KUKA KRL program: EPS_2_25252_SD3A_A_20250910061721.src

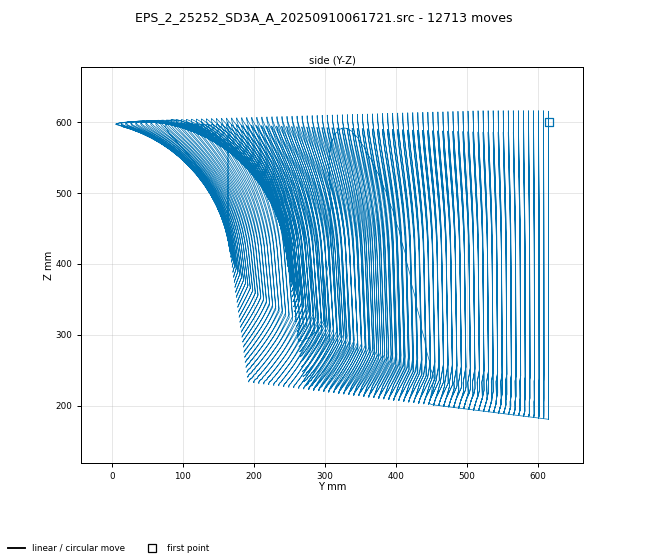
[picture p0: tool path of EPS_2_25252_SD3A_A_20250910061721.src, 12713 of 12715 moves have a stored position in this frame; points joined in program order, loops and branches not executed]
&ACCESS RVP
&REL 4
&COMMENT QRS 19112012
&PARAM EDITMASK = *
DEF PART()
EXT BAS (BAS_COMMAND :IN,REAL :IN )
INT I
BAS (#INITMOV,0 )

;KUKA QRS Post kuka4.cps  Date:22-06-2017 !

File_ID=2824

QRS_PRE_INIT()

;Init var - Until changes are made in qrs_pre_init
Outlet_Square_prg=0
Inlet_1_Square_prg=0
Inlet_2_Square_prg=0
Inlet_3_Square_prg=0
Inlet_4_Square_prg=0
Inlet_5_Square_prg=0

Outlet_1={X 0.000, Y 518.380, Z 433.000, B 0.000, E1 0.000 }
Inlet_1={X 0.000, Y 520.620, Z 403.000, B 0.000, E1 207.000 }
Outlet_1_type=366
Inlet_1_type=366
;QRS#1=Sidecore dimensions
;QRS#2=375-15" PVC SDR 35
;QRS#3=375-15" PVC SDR 35
;QRS#4=
;QRS#5=
;QRS#6=
;QRS#7=
;QRS#8=
;QRS#9=20Y PSX
;QRS#10=20Y PSX
;QRS#11=
;QRS#12=
;QRS#13=
;QRS#14=
;QRS#15=
;QRS#16=1220x127x914 3'
;QRS#17=EPS Height
;QRS#18=616
;QRS#19=*
;QRS#20= UPDATED VERSION 22-06-2017
;QRS#21=*
Outlet_Square=0250
Inlet_1_Square=0250
Inlet_2_Square=0
Inlet_3_Square=0
Inlet_4_Square=0
Inlet_5_Square=0
Mill_Square=1
Outlet_Square_Prg=252
Inlet_1_Square_prg=252

QRS_INIT()

$ADVANCE=5

; T1
PTP {E1 173.576,E2 173.576}
PTP {X 0,Y 615.507,A -85,B 0,C 180,E1 173.576,E2 173.576,E3 0,E4 0,E5 0,E6 0}
QRS_SPEED_INIT()
LIN {X 0,Y 615.507,Z 600,A -85,B 0,C 180,E1 173.576,E2 173.576,E3 0,E4 0,E5 0,E6 0} C_VEL
LIN {X 0,Y 615.507,Z 191.184,A -85,B 0,C 180,E1 173.576,E2 173.576} C_VEL
LIN {X 0,Y 615.507,Z 183.015,A -85,B 0,C 180,E1 173.576,E2 173.576} C_VEL
LIN {X 0,Y 615.486,Z 181.015,A -85,B 0,C 180,E1 173.39,E2 173.39} C_VEL
LIN {X 0,Y 615.462,Z 181.004,A -85,B 0,C 180,E1 170.8,E2 170.8} C_VEL
LIN {X 0,Y 615.46,Z 181.004,A -85,B 0,C 180,E1 168.806,E2 168.806} C_VEL
LIN {X 0,Y 615.457,Z 181.004,A -85,B 0,C 180,E1 166.798,E2 166.798} C_VEL
LIN {X 0,Y 615.453,Z 181.004,A -85,B 0,C 180,E1 164.773,E2 164.773} C_VEL
LIN {X 0,Y 615.448,Z 181.005,A -85,B 0,C 180,E1 162.728,E2 162.728} C_VEL
LIN {X 0,Y 615.442,Z 181.006,A -85,B 0,C 180,E1 160.66,E2 160.66} C_VEL
LIN {X 0,Y 615.437,Z 181.006,A -85,B 0,C 180,E1 158.566,E2 158.566} C_VEL
LIN {X 0,Y 615.45,Z 181.01,A -85,B 0,C 180,E1 155.991,E2 155.991} C_VEL
LIN {X 0,Y 615.495,Z 181.013,A -85,B 0,C 180,E1 153.556,E2 153.556} C_VEL
LIN {X 0,Y 615.489,Z 181.006,A -85,B 0,C 180,E1 151.342,E2 151.342} C_VEL
LIN {X 0,Y 615.45,Z 181.005,A -85,B 0,C 180,E1 148.913,E2 148.913} C_VEL
LIN {X 0,Y 615.432,Z 181.008,A -85,B 0,C 180,E1 146.467,E2 146.467} C_VEL
LIN {X 0,Y 615.445,Z 181.01,A -85,B 0,C 180,E1 144.166,E2 144.166} C_VEL
LIN {X 0,Y 615.47,Z 181.011,A -85,B 0,C 180,E1 141.93,E2 141.93} C_VEL
LIN {X 0,Y 615.488,Z 181.004,A -85,B 0,C 180,E1 139.393,E2 139.393} C_VEL
LIN {X 0,Y 615.434,Z 181.007,A -85,B 0,C 180,E1 136.75,E2 136.75} C_VEL
LIN {X 0,Y 615.467,Z 181.012,A -85,B 0,C 180,E1 133.995,E2 133.995} C_VEL
LIN {X 0,Y 615.448,Z 181.005,A -85,B 0,C 180,E1 131.09,E2 131.09} C_VEL
LIN {X 0,Y 615.433,Z 181.007,A -85,B 0,C 180,E1 128.905,E2 128.905} C_VEL
LIN {X 0,Y 615.44,Z 181.009,A -85,B 0,C 180,E1 126.424,E2 126.424} C_VEL
LIN {X 0,Y 615.477,Z 181.013,A -85,B 0,C 180,E1 124.019,E2 124.019} C_VEL
LIN {X 0,Y 615.439,Z 181.006,A -85,B 0,C 180,E1 121.078,E2 121.078} C_VEL
LIN {X 0,Y 615.434,Z 181.009,A -85,B 0,C 180,E1 118.658,E2 118.658} C_VEL
LIN {X 0,Y 615.499,Z 181.003,A -85,B 0,C 180,E1 115.712,E2 115.712} C_VEL
LIN {X 0,Y 615.474,Z 181.004,A -85,B 0,C 180,E1 113.554,E2 113.554} C_VEL
LIN {X 0,Y 615.456,Z 181.005,A -85,B 0,C 180,E1 111.43,E2 111.43} C_VEL
LIN {X 0,Y 615.447,Z 181.006,A -85,B 0,C 180,E1 109.337,E2 109.337} C_VEL
LIN {X 0,Y 615.441,Z 181.006,A -85,B 0,C 180,E1 107.269,E2 107.269} C_VEL
LIN {X 0,Y 615.437,Z 181.007,A -85,B 0,C 180,E1 105.225,E2 105.225} C_VEL
LIN {X 0,Y 615.435,Z 181.007,A -85,B 0,C 180,E1 103.2,E2 103.2} C_VEL
LIN {X 0,Y 615.432,Z 181.009,A -85,B 0,C 180,E1 100.859,E2 100.859} C_VEL
LIN {X 0,Y 615.452,Z 181.011,A -85,B 0,C 180,E1 98.535,E2 98.535} C_VEL
LIN {X 0,Y 615.493,Z 181.004,A -85,B 0,C 180,E1 95.897,E2 95.897} C_VEL
LIN {X 0,Y 615.433,Z 181.007,A -85,B 0,C 180,E1 93.272,E2 93.272} C_VEL
LIN {X 0,Y 615.433,Z 181.007,A -85,B 0,C 180,E1 91.307,E2 91.307} C_VEL
LIN {X 0,Y 615.434,Z 181.007,A -85,B 0,C 180,E1 89.344,E2 89.344} C_VEL
LIN {X 0,Y 615.429,Z 181.112,A -85,B 0,C 180,E1 87.237,E2 87.237} C_VEL
LIN {X 0,Y 615.455,Z 205.741,A -85,B 0,C 180,E1 84.983,E2 84.983} C_VEL
LIN {X 0,Y 615.489,Z 392.91,A -85,B 0,C 180,E1 82.68,E2 82.68} C_VEL
LIN {X 0,Y 615.492,Z 415.248,A -85,B 0,C 180,E1 82.371,E2 82.371} C_VEL
LIN {X 0,Y 615.494,Z 430.502,A -85,B 0,C 180,E1 82.041,E2 82.041} C_VEL
LIN {X 0,Y 615.492,Z 446.908,A -85,B 0,C 180,E1 81.545,E2 81.545} C_VEL
LIN {X 0,Y 615.491,Z 461.835,A -85,B 0,C 180,E1 80.966,E2 80.966} C_VEL
LIN {X 0,Y 615.492,Z 475.89,A -85,B 0,C 180,E1 80.303,E2 80.303} C_VEL
LIN {X 0,Y 615.498,Z 490.392,A -85,B 0,C 180,E1 79.472,E2 79.472} C_VEL
LIN {X 0,Y 615.497,Z 503.871,A -85,B 0,C 180,E1 78.556,E2 78.556} C_VEL
LIN {X 0,Y 615.495,Z 517.429,A -85,B 0,C 180,E1 77.469,E2 77.469} C_VEL
LIN {X 0,Y 615.496,Z 529.84,A -85,B 0,C 180,E1 76.293,E2 76.293} C_VEL
LIN {X 0,Y 615.489,Z 540.486,A -85,B 0,C 180,E1 75.112,E2 75.112} C_VEL
LIN {X 0,Y 615.495,Z 550.328,A -85,B 0,C 180,E1 73.832,E2 73.832} C_VEL
LIN {X 0,Y 615.493,Z 558.546,A -85,B 0,C 180,E1 72.557,E2 72.557} C_VEL
LIN {X 0,Y 615.489,Z 565.176,A -85,B 0,C 180,E1 71.353,E2 71.353} C_VEL
LIN {X 0,Y 615.496,Z 571.501,A -85,B 0,C 180,E1 69.967,E2 69.967} C_VEL
LIN {X 0,Y 615.484,Z 576.552,A -85,B 0,C 180,E1 68.567,E2 68.567} C_VEL
LIN {X 0,Y 615.484,Z 580.491,A -85,B 0,C 180,E1 67.155,E2 67.155} C_VEL
LIN {X 0,Y 615.487,Z 583.245,A -85,B 0,C 180,E1 65.727,E2 65.727} C_VEL
LIN {X 0,Y 615.5,Z 584.853,A -85,B 0,C 180,E1 64.284,E2 64.284} C_VEL
LIN {X 0,Y 615.493,Z 585.363,A -85,B 0,C 180,E1 62.822,E2 62.822} C_VEL
LIN {X 0,Y 615.486,Z 584.657,A -85,B 0,C 180,E1 61.341,E2 61.341} C_VEL
LIN {X 0,Y 615.494,Z 582.669,A -85,B 0,C 180,E1 59.84,E2 59.84} C_VEL
LIN {X 0,Y 615.491,Z 579.372,A -85,B 0,C 180,E1 58.314,E2 58.314} C_VEL
LIN {X 0,Y 615.487,Z 575.946,A -85,B 0,C 180,E1 57.154,E2 57.154} C_VEL
LIN {X 0,Y 615.489,Z 570.196,A -85,B 0,C 180,E1 55.639,E2 55.639} C_VEL
LIN {X 0,Y 615.495,Z 563.135,A -85,B 0,C 180,E1 54.166,E2 54.166} C_VEL
LIN {X 0,Y 615.491,Z 554.897,A -85,B 0,C 180,E1 52.758,E2 52.758} C_VEL
LIN {X 0,Y 615.495,Z 546.174,A -85,B 0,C 180,E1 51.515,E2 51.515} C_VEL
LIN {X 0,Y 615.494,Z 535.742,A -85,B 0,C 180,E1 50.25,E2 50.25} C_VEL
LIN {X 0,Y 615.492,Z 523.889,A -85,B 0,C 180,E1 49.028,E2 49.028} C_VEL
LIN {X 0,Y 615.493,Z 511.215,A -85,B 0,C 180,E1 47.92,E2 47.92} C_VEL
LIN {X 0,Y 615.494,Z 498.258,A -85,B 0,C 180,E1 46.953,E2 46.953} C_VEL
LIN {X 0,Y 615.496,Z 484.758,A -85,B 0,C 180,E1 46.097,E2 46.097} C_VEL
LIN {X 0,Y 615.491,Z 468.938,A -85,B 0,C 180,E1 45.265,E2 45.265} C_VEL
LIN {X 0,Y 615.495,Z 454.323,A -85,B 0,C 180,E1 44.637,E2 44.637} C_VEL
LIN {X 0,Y 615.491,Z 439.135,A -85,B 0,C 180,E1 44.112,E2 44.112} C_VEL
LIN {X 0,Y 615.496,Z 422.955,A -85,B 0,C 180,E1 43.69,E2 43.69} C_VEL
LIN {X 0,Y 615.491,Z 407.024,A -85,B 0,C 180,E1 43.409,E2 43.409} C_VEL
LIN {X 0,Y 615.482,Z 205.725,A -85,B 0,C 180,E1 40.927,E2 40.927} C_VEL
LIN {X 0,Y 615.492,Z 180.994,A -85,B 0,C 180,E1 38.642,E2 38.642} C_VEL
LIN {X 0,Y 615.493,Z 181.011,A -85,B 0,C 180,E1 35.616,E2 35.616} C_VEL
LIN {X 0,Y 615.472,Z 181.004,A -85,B 0,C 180,E1 33.238,E2 33.238} C_VEL
LIN {X 0,Y 615.48,Z 180.997,A -85,B 0,C 180,E1 30.921,E2 30.921} C_VEL
LIN {X 0,Y 615.486,Z 180.998,A -85,B 0,C 180,E1 28.451,E2 28.451} C_VEL
LIN {X 0,Y 615.477,Z 181.008,A -85,B 0,C 180,E1 25.568,E2 25.568} C_VEL
LIN {X 0,Y 615.49,Z 180.994,A -85,B 0,C 180,E1 22.845,E2 22.845} C_VEL
LIN {X 0,Y 615.486,Z 181.013,A -85,B 0,C 180,E1 20.033,E2 20.033} C_VEL
LIN {X 0,Y 615.469,Z 181.001,A -85,B 0,C 180,E1 17.271,E2 17.271} C_VEL
LIN {X 0,Y 615.487,Z 181,A -85,B 0,C 180,E1 14.549,E2 14.549} C_VEL
LIN {X 0,Y 615.48,Z 181.009,A -85,B 0,C 180,E1 11.861,E2 11.861} C_VEL
LIN {X 0,Y 615.473,Z 180.998,A -85,B 0,C 180,E1 9.199,E2 9.199} C_VEL
LIN {X 0,Y 615.487,Z 181.003,A -85,B 0,C 180,E1 6.557,E2 6.557} C_VEL
LIN {X 0,Y 615.474,Z 181.008,A -85,B 0,C 180,E1 3.929,E2 3.929} C_VEL
LIN {X 0,Y 615.472,Z 180.999,A -85,B 0,C 180,E1 1.309,E2 1.309} C_VEL
LIN {X 0,Y 615.489,Z 181.003,A -85,B 0,C 180,E1 -1.308,E2 -1.308} C_VEL
LIN {X 0,Y 615.473,Z 181.009,A -85,B 0,C 180,E1 -3.928,E2 -3.928} C_VEL
LIN {X 0,Y 615.469,Z 180.999,A -85,B 0,C 180,E1 -6.569,E2 -6.569} C_VEL
LIN {X 0,Y 615.49,Z 181.003,A -85,B 0,C 180,E1 -9.198,E2 -9.198} C_VEL
LIN {X 0,Y 615.469,Z 181.008,A -85,B 0,C 180,E1 -11.861,E2 -11.861} C_VEL
LIN {X 0,Y 615.472,Z 180.999,A -85,B 0,C 180,E1 -14.549,E2 -14.549} C_VEL
LIN {X 0,Y 615.493,Z 181.008,A -85,B 0,C 180,E1 -17.27,E2 -17.27} C_VEL
LIN {X 0,Y 615.454,Z 181.005,A -85,B 0,C 180,E1 -20.034,E2 -20.034} C_VEL
LIN {X 0,Y 615.463,Z 181.001,A -85,B 0,C 180,E1 -22.342,E2 -22.342} C_VEL
LIN {X 0,Y 615.492,Z 181.004,A -85,B 0,C 180,E1 -24.991,E2 -24.991} C_VEL
LIN {X 0,Y 615.453,Z 181.005,A -85,B 0,C 180,E1 -27.916,E2 -27.916} C_VEL
LIN {X 0,Y 615.455,Z 181.002,A -85,B 0,C 180,E1 -30.162,E2 -30.162} C_VEL
LIN {X 0,Y 615.479,Z 180.998,A -85,B 0,C 180,E1 -32.458,E2 -32.458} C_VEL
LIN {X 0,Y 615.492,Z 181.003,A -85,B 0,C 180,E1 -34.814,E2 -34.814} C_VEL
LIN {X 0,Y 615.483,Z 181.011,A -85,B 0,C 180,E1 -37.242,E2 -37.242} C_VEL
LIN {X 0,Y 615.449,Z 181.006,A -85,B 0,C 180,E1 -39.753,E2 -39.753} C_VEL
LIN {X 0,Y 615.478,Z 180.999,A -85,B 0,C 180,E1 -42.353,E2 -42.353} C_VEL
LIN {X 0,Y 615.487,Z 181.012,A -85,B 0,C 180,E1 -45.068,E2 -45.068} C_VEL
LIN {X 0,Y 615.446,Z 181.006,A -85,B 0,C 180,E1 -47.643,E2 -47.643} C_VEL
LIN {X 0,Y 615.476,Z 181,A -85,B 0,C 180,E1 -50.249,E2 -50.249} C_VEL
LIN {X 0,Y 615.472,Z 181.011,A -85,B 0,C 180,E1 -53.065,E2 -53.065} C_VEL
LIN {X 0,Y 615.45,Z 181.008,A -85,B 0,C 180,E1 -55.304,E2 -55.304} C_VEL
LIN {X 0,Y 615.443,Z 181.005,A -85,B 0,C 180,E1 -57.675,E2 -57.675} C_VEL
LIN {X 0,Y 615.482,Z 181.001,A -85,B 0,C 180,E1 -60.206,E2 -60.206} C_VEL
LIN {X 0,Y 615.465,Z 181.01,A -85,B 0,C 180,E1 -62.959,E2 -62.959} C_VEL
LIN {X 0,Y 615.441,Z 181.176,A -85,B 0,C 180,E1 -63.599,E2 -63.599} C_VEL
LIN {X 0,Y 615.497,Z 213.161,A -85,B 0,C 180,E1 -66.217,E2 -66.217} C_VEL
LIN {X 0,Y 615.485,Z 235.002,A -85,B 0,C 180,E1 -67.973,E2 -67.973} C_VEL
LIN {X 0,Y 615.49,Z 442.374,A -85,B 0,C 180,E1 -70.531,E2 -70.531} C_VEL
LIN {X 0,Y 615.493,Z 458.958,A -85,B 0,C 180,E1 -70.878,E2 -70.878} C_VEL
LIN {X 0,Y 615.493,Z 473.906,A -85,B 0,C 180,E1 -71.31,E2 -71.31} C_VEL
LIN {X 0,Y 615.492,Z 489.332,A -85,B 0,C 180,E1 -71.88,E2 -71.88} C_VEL
LIN {X 0,Y 615.493,Z 503.986,A -85,B 0,C 180,E1 -72.557,E2 -72.557} C_VEL
LIN {X 0,Y 615.5,Z 517.82,A -85,B 0,C 180,E1 -73.327,E2 -73.327} C_VEL
LIN {X 0,Y 615.499,Z 532.024,A -85,B 0,C 180,E1 -74.264,E2 -74.264} C_VEL
LIN {X 0,Y 615.495,Z 545.08,A -85,B 0,C 180,E1 -75.281,E2 -75.281} C_VEL
LIN {X 0,Y 615.494,Z 556.202,A -85,B 0,C 180,E1 -76.293,E2 -76.293} C_VEL
LIN {X 0,Y 615.493,Z 567.281,A -85,B 0,C 180,E1 -77.469,E2 -77.469} C_VEL
LIN {X 0,Y 615.495,Z 576.758,A -85,B 0,C 180,E1 -78.639,E2 -78.639} C_VEL
LIN {X 0,Y 615.496,Z 585.957,A -85,B 0,C 180,E1 -79.971,E2 -79.971} C_VEL
LIN {X 0,Y 615.489,Z 594.495,A -85,B 0,C 180,E1 -81.462,E2 -81.462} C_VEL
LIN {X 0,Y 615.491,Z 601.979,A -85,B 0,C 180,E1 -83.101,E2 -83.101} C_VEL
LIN {X 0,Y 615.492,Z 607.737,A -85,B 0,C 180,E1 -84.757,E2 -84.757} C_VEL
LIN {X 0,Y 615.493,Z 611.073,A -85,B 0,C 180,E1 -86.07,E2 -86.07} C_VEL
LIN {X 0,Y 615.485,Z 613.502,A -85,B 0,C 180,E1 -87.381,E2 -87.381} C_VEL
LIN {X 0,Y 615.488,Z 614.869,A -85,B 0,C 180,E1 -88.69,E2 -88.69} C_VEL
LIN {X 0,Y 615.489,Z 615.39,A -85,B 0,C 180,E1 -89.998,E2 -89.998} C_VEL
LIN {X 0,Y 615.488,Z 614.871,A -85,B 0,C 180,E1 -91.307,E2 -91.307} C_VEL
LIN {X 0,Y 615.485,Z 613.507,A -85,B 0,C 180,E1 -92.616,E2 -92.616} C_VEL
LIN {X 0,Y 615.493,Z 611.08,A -85,B 0,C 180,E1 -93.927,E2 -93.927} C_VEL
LIN {X 0,Y 615.492,Z 607.747,A -85,B 0,C 180,E1 -95.239,E2 -95.239} C_VEL
LIN {X 0,Y 615.491,Z 601.986,A -85,B 0,C 180,E1 -96.897,E2 -96.897} C_VEL
LIN {X 0,Y 615.489,Z 594.511,A -85,B 0,C 180,E1 -98.535,E2 -98.535} C_VEL
LIN {X 0,Y 615.496,Z 585.976,A -85,B 0,C 180,E1 -100.026,E2 -100.026} C_VEL
LIN {X 0,Y 615.494,Z 576.781,A -85,B 0,C 180,E1 -101.358,E2 -101.358} C_VEL
LIN {X 0,Y 615.495,Z 567.309,A -85,B 0,C 180,E1 -102.528,E2 -102.528} C_VEL
LIN {X 0,Y 615.496,Z 556.236,A -85,B 0,C 180,E1 -103.703,E2 -103.703} C_VEL
LIN {X 0,Y 615.495,Z 544.141,A -85,B 0,C 180,E1 -104.8,E2 -104.8} C_VEL
LIN {X 0,Y 615.498,Z 530.909,A -85,B 0,C 180,E1 -105.818,E2 -105.818} C_VEL
LIN {X 0,Y 615.5,Z 517.874,A -85,B 0,C 180,E1 -106.669,E2 -106.669} C_VEL
LIN {X 0,Y 615.493,Z 504.053,A -85,B 0,C 180,E1 -107.439,E2 -107.439} C_VEL
LIN {X 0,Y 615.491,Z 489.389,A -85,B 0,C 180,E1 -108.118,E2 -108.118} C_VEL
LIN {X 0,Y 615.493,Z 474.005,A -85,B 0,C 180,E1 -108.687,E2 -108.687} C_VEL
LIN {X 0,Y 615.498,Z 457.273,A -85,B 0,C 180,E1 -109.162,E2 -109.162} C_VEL
LIN {X 0,Y 615.49,Z 441.11,A -85,B 0,C 180,E1 -109.487,E2 -109.487} C_VEL
LIN {X 0,Y 615.485,Z 235.044,A -85,B 0,C 180,E1 -112.024,E2 -112.024} C_VEL
LIN {X 0,Y 615.453,Z 201.645,A -85,B 0,C 180,E1 -114.72,E2 -114.72} C_VEL
LIN {X 0,Y 615.44,Z 181.006,A -85,B 0,C 180,E1 -116.421,E2 -116.421} C_VEL
LIN {X 0,Y 615.441,Z 181.008,A -85,B 0,C 180,E1 -118.657,E2 -118.657} C_VEL
LIN {X 0,Y 615.472,Z 181.011,A -85,B 0,C 180,E1 -121.084,E2 -121.084} C_VEL
LIN {X 0,Y 615.455,Z 181.003,A -85,B 0,C 180,E1 -124.021,E2 -124.021} C_VEL
LIN {X 0,Y 615.438,Z 181.007,A -85,B 0,C 180,E1 -126.425,E2 -126.425} C_VEL
LIN {X 0,Y 615.479,Z 181.011,A -85,B 0,C 180,E1 -129.062,E2 -129.062} C_VEL
LIN {X 0,Y 615.495,Z 181.004,A -85,B 0,C 180,E1 -131.469,E2 -131.469} C_VEL
LIN {X 0,Y 615.441,Z 181.005,A -85,B 0,C 180,E1 -134.149,E2 -134.149} C_VEL
LIN {X 0,Y 615.476,Z 181.011,A -85,B 0,C 180,E1 -136.949,E2 -136.949} C_VEL
LIN {X 0,Y 615.45,Z 181.004,A -85,B 0,C 180,E1 -139.91,E2 -139.91} C_VEL
LIN {X 0,Y 615.444,Z 181.005,A -85,B 0,C 180,E1 -141.988,E2 -141.988} C_VEL
LIN {X 0,Y 615.439,Z 181.008,A -85,B 0,C 180,E1 -144.381,E2 -144.381} C_VEL
LIN {X 0,Y 615.466,Z 181.011,A -85,B 0,C 180,E1 -146.763,E2 -146.763} C_VEL
LIN {X 0,Y 615.491,Z 181.012,A -85,B 0,C 180,E1 -149.081,E2 -149.081} C_VEL
LIN {X 0,Y 615.469,Z 181.003,A -85,B 0,C 180,E1 -151.545,E2 -151.545} C_VEL
LIN {X 0,Y 615.462,Z 181.004,A -85,B 0,C 180,E1 -153.555,E2 -153.555} C_VEL
LIN {X 0,Y 615.437,Z 181.006,A -85,B 0,C 180,E1 -155.993,E2 -155.993} C_VEL
LIN {X 0,Y 615.441,Z 181.005,A -85,B 0,C 180,E1 -157.862,E2 -157.862} C_VEL
LIN {X 0,Y 615.434,Z 181.007,A -85,B 0,C 180,E1 -159.966,E2 -159.966} C_VEL
LIN {X 0,Y 615.478,Z 181.012,A -85,B 0,C 180,E1 -162.73,E2 -162.73} C_VEL
LIN {X 0,Y 615.464,Z 181.003,A -85,B 0,C 180,E1 -165.451,E2 -165.451} C_VEL
LIN {X 0,Y 615.46,Z 181.004,A -85,B 0,C 180,E1 -167.47,E2 -167.47} C_VEL
LIN {X 0,Y 615.457,Z 181.004,A -85,B 0,C 180,E1 -169.473,E2 -169.473} C_VEL
LIN {X 0,Y 615.452,Z 181.005,A -85,B 0,C 180,E1 -171.463,E2 -171.463} C_VEL
LIN {X 0,Y 615.456,Z 181.004,A -85,B 0,C 180,E1 -173.443,E2 -173.443} C_VEL
LIN {X 0,Y 615.456,Z 181.004,A -85,B 0,C 180,E1 -175.416,E2 -175.416} C_VEL
LIN {X 0,Y 615.457,Z 181.004,A -85,B 0,C 180,E1 -177.382,E2 -177.382} C_VEL
LIN {X 0,Y 615.459,Z 181.004,A -85,B 0,C 180,E1 -179.346,E2 -179.346} C_VEL
LIN {X 0,Y 615.46,Z 181.004,A -85,B 0,C 180,E1 -181.309,E2 -181.309} C_VEL
LIN {X 0,Y 615.436,Z 181.008,A -85,B 0,C 180,E1 -183.929,E2 -183.929} C_VEL
LIN {X 0,Y 615.486,Z 181.015,A -85,B 0,C 180,E1 -186.61,E2 -186.61} C_VEL
LIN {X 0,Y 614.795,Z 181.151,A -85,B 0,C 180,E1 -187.156,E2 -187.156} C_VEL
LIN {X 0,Y 611.95,Z 181.566,A -85,B 0,C 180,E1 -188.042,E2 -188.042} C_VEL
LIN {X 0,Y 609.555,Z 181.875,A -85,B 0,C 180,E1 -188.754,E2 -188.754} C_VEL
LIN {X 0,Y 608.517,Z 181.993,A -85,B 0,C 180,E1 -189.304,E2 -189.304} C_VEL
LIN {X 0,Y 608.425,Z 182.003,A -85,B 0,C 180,E1 -189.49,E2 -189.49} C_VEL
LIN {X 0,Y 608.423,Z 182.005,A -85,B 0,C 180,E1 -192.001,E2 -192.001} C_VEL
LIN {X 0,Y 608.465,Z 182.006,A -85,B 0,C 180,E1 -194.721,E2 -194.721} C_VEL
LIN {X 0,Y 608.459,Z 182.005,A -85,B 0,C 180,E1 -196.784,E2 -196.784} C_VEL
LIN {X 0,Y 608.411,Z 182.005,A -85,B 0,C 180,E1 -199.572,E2 -199.572} C_VEL
LIN {X 0,Y 608.429,Z 182.003,A -85,B 0,C 180,E1 -201.693,E2 -201.693} C_VEL
LIN {X 0,Y 608.436,Z 182.01,A -85,B 0,C 180,E1 -204.572,E2 -204.572} C_VEL
LIN {X 0,Y 608.411,Z 182.005,A -85,B 0,C 180,E1 -207.52,E2 -207.52} C_VEL
LIN {X 0,Y 608.431,Z 182.006,A -85,B 0,C 180,E1 -209.973,E2 -209.973} C_VEL
LIN {X 0,Y 608.435,Z 182.004,A -85,B 0,C 180,E1 -212.881,E2 -212.881} C_VEL
LIN {X 0,Y 608.406,Z 182.006,A -85,B 0,C 180,E1 -215.281,E2 -215.281} C_VEL
LIN {X 0,Y 608.439,Z 182.004,A -85,B 0,C 180,E1 -217.749,E2 -217.749} C_VEL
LIN {X 0,Y 608.46,Z 182.009,A -85,B 0,C 180,E1 -220.335,E2 -220.335} C_VEL
LIN {X 0,Y 608.416,Z 182.005,A -85,B 0,C 180,E1 -222.964,E2 -222.964} C_VEL
LIN {X 0,Y 608.411,Z 182.005,A -85,B 0,C 180,E1 -225.204,E2 -225.204} C_VEL
LIN {X 0,Y 608.443,Z 182.007,A -85,B 0,C 180,E1 -227.941,E2 -227.941} C_VEL
LIN {X 0,Y 608.42,Z 182.006,A -85,B 0,C 180,E1 -230.709,E2 -230.709} C_VEL
LIN {X 0,Y 608.407,Z 182.005,A -85,B 0,C 180,E1 -233.085,E2 -233.085} C_VEL
LIN {X 0,Y 608.432,Z 182.004,A -85,B 0,C 180,E1 -235.532,E2 -235.532} C_VEL
LIN {X 0,Y 608.445,Z 182.008,A -85,B 0,C 180,E1 -237.908,E2 -237.908} C_VEL
LIN {X 0,Y 608.48,Z 182.004,A -85,B 0,C 180,E1 -240.224,E2 -240.224} C_VEL
LIN {X 0,Y 608.403,Z 182.006,A -85,B 0,C 180,E1 -243.226,E2 -243.226} C_VEL
LIN {X 0,Y 608.422,Z 182.006,A -85,B 0,C 180,E1 -245.43,E2 -245.43} C_VEL
LIN {X 0,Y 608.45,Z 182.005,A -85,B 0,C 180,E1 -248.31,E2 -248.31} C_VEL
LIN {X 0,Y 608.427,Z 182.003,A -85,B 0,C 180,E1 -251.132,E2 -251.132} C_VEL
LIN {X 0,Y 608.453,Z 182.011,A -85,B 0,C 180,E1 -253.908,E2 -253.908} C_VEL
LIN {X 0,Y 608.43,Z 182.003,A -85,B 0,C 180,E1 -256.645,E2 -256.645} C_VEL
LIN {X 0,Y 608.425,Z 182.006,A -85,B 0,C 180,E1 -259.352,E2 -259.352} C_VEL
LIN {X 0,Y 608.473,Z 182.005,A -85,B 0,C 180,E1 -262.035,E2 -262.035} C_VEL
LIN {X 0,Y 608.421,Z 182.004,A -85,B 0,C 180,E1 -264.7,E2 -264.7} C_VEL
LIN {X 0,Y 608.444,Z 182.005,A -85,B 0,C 180,E1 -267.354,E2 -267.354} C_VEL
LIN {X 0,Y 608.477,Z 182.004,A -85,B 0,C 180,E1 -270.002,E2 -270.002} C_VEL
LIN {X 0,Y 608.436,Z 182.197,A -85,B 0,C 180,E1 -272.567,E2 -272.567} C_VEL
LIN {X 0,Y 608.717,Z 193.625,A -85,B 0,C 180,E1 -273.642,E2 -273.642} C_VEL
LIN {X 0,Y 608.636,Z 205.796,A -85,B 0,C 180,E1 -274.762,E2 -274.762} C_VEL
LIN {X 0,Y 608.876,Z 210.931,A -85,B 0,C 180,E1 -274.843,E2 -274.843} C_VEL
LIN {X 0,Y 608.815,Z 411.348,A -85,B 0,C 180,E1 -277.338,E2 -277.338} C_VEL
LIN {X 0,Y 608.775,Z 427.683,A -85,B 0,C 180,E1 -277.672,E2 -277.672} C_VEL
LIN {X 0,Y 608.754,Z 443.666,A -85,B 0,C 180,E1 -278.132,E2 -278.132} C_VEL
LIN {X 0,Y 608.703,Z 459.382,A -85,B 0,C 180,E1 -278.717,E2 -278.717} C_VEL
LIN {X 0,Y 608.66,Z 475.413,A -85,B 0,C 180,E1 -279.472,E2 -279.472} C_VEL
LIN {X 0,Y 608.629,Z 490.001,A -85,B 0,C 180,E1 -280.312,E2 -280.312} C_VEL
LIN {X 0,Y 608.585,Z 503.661,A -85,B 0,C 180,E1 -281.246,E2 -281.246} C_VEL
LIN {X 0,Y 608.544,Z 517.201,A -85,B 0,C 180,E1 -282.338,E2 -282.338} C_VEL
LIN {X 0,Y 608.497,Z 529.711,A -85,B 0,C 180,E1 -283.527,E2 -283.527} C_VEL
LIN {X 0,Y 608.486,Z 540.445,A -85,B 0,C 180,E1 -284.721,E2 -284.721} C_VEL
LIN {X 0,Y 608.458,Z 550.929,A -85,B 0,C 180,E1 -286.095,E2 -286.095} C_VEL
LIN {X 0,Y 608.469,Z 559.727,A -85,B 0,C 180,E1 -287.477,E2 -287.477} C_VEL
LIN {X 0,Y 608.443,Z 567.104,A -85,B 0,C 180,E1 -288.871,E2 -288.871} C_VEL
LIN {X 0,Y 608.438,Z 573.211,A -85,B 0,C 180,E1 -290.276,E2 -290.276} C_VEL
LIN {X 0,Y 608.426,Z 578.09,A -85,B 0,C 180,E1 -291.694,E2 -291.694} C_VEL
LIN {X 0,Y 608.427,Z 581.751,A -85,B 0,C 180,E1 -293.126,E2 -293.126} C_VEL
LIN {X 0,Y 608.406,Z 584.315,A -85,B 0,C 180,E1 -294.574,E2 -294.574} C_VEL
LIN {X 0,Y 608.42,Z 585.7,A -85,B 0,C 180,E1 -296.037,E2 -296.037} C_VEL
LIN {X 0,Y 608.425,Z 585.894,A -85,B 0,C 180,E1 -297.52,E2 -297.52} C_VEL
LIN {X 0,Y 608.407,Z 584.897,A -85,B 0,C 180,E1 -299.024,E2 -299.024} C_VEL
LIN {X 0,Y 608.43,Z 582.651,A -85,B 0,C 180,E1 -300.548,E2 -300.548} C_VEL
LIN {X 0,Y 608.417,Z 578.946,A -85,B 0,C 180,E1 -302.098,E2 -302.098} C_VEL
LIN {X 0,Y 608.425,Z 573.535,A -85,B 0,C 180,E1 -303.727,E2 -303.727} C_VEL
LIN {X 0,Y 608.43,Z 566.815,A -85,B 0,C 180,E1 -305.279,E2 -305.279} C_VEL
LIN {X 0,Y 608.471,Z 559.156,A -85,B 0,C 180,E1 -306.708,E2 -306.708} C_VEL
LIN {X 0,Y 608.48,Z 550.942,A -85,B 0,C 180,E1 -307.993,E2 -307.993} C_VEL
LIN {X 0,Y 608.483,Z 541.012,A -85,B 0,C 180,E1 -309.298,E2 -309.298} C_VEL
LIN {X 0,Y 608.508,Z 530.16,A -85,B 0,C 180,E1 -310.516,E2 -310.516} C_VEL
LIN {X 0,Y 608.547,Z 518.193,A -85,B 0,C 180,E1 -311.665,E2 -311.665} C_VEL
LIN {X 0,Y 608.573,Z 505.702,A -85,B 0,C 180,E1 -312.693,E2 -312.693} C_VEL
LIN {X 0,Y 608.611,Z 492.473,A -85,B 0,C 180,E1 -313.624,E2 -313.624} C_VEL
LIN {X 0,Y 608.643,Z 478.411,A -85,B 0,C 180,E1 -314.455,E2 -314.455} C_VEL
LIN {X 0,Y 608.689,Z 462.722,A -85,B 0,C 180,E1 -315.225,E2 -315.225} C_VEL
LIN {X 0,Y 608.73,Z 446.825,A -85,B 0,C 180,E1 -315.852,E2 -315.852} C_VEL
LIN {X 0,Y 608.768,Z 430.544,A -85,B 0,C 180,E1 -316.349,E2 -316.349} C_VEL
LIN {X 0,Y 608.801,Z 413.508,A -85,B 0,C 180,E1 -316.717,E2 -316.717} C_VEL
LIN {X 0,Y 608.821,Z 376.219,A -85,B 0,C 180,E1 -317.2,E2 -317.2} C_VEL
LIN {X 0,Y 608.878,Z 206.999,A -85,B 0,C 180,E1 -319.296,E2 -319.296} C_VEL
LIN {X 0,Y 608.692,Z 205.634,A -85,B 0,C 180,E1 -319.341,E2 -319.341} C_VEL
LIN {X 0,Y 608.709,Z 183.074,A -85,B 0,C 180,E1 -321.429,E2 -321.429} C_VEL
LIN {X 0,Y 608.463,Z 182.001,A -85,B 0,C 180,E1 -321.552,E2 -321.552} C_VEL
LIN {X 0,Y 608.462,Z 182.004,A -85,B 0,C 180,E1 -323.952,E2 -323.952} C_VEL
LIN {X 0,Y 608.45,Z 182.01,A -85,B 0,C 180,E1 -326.328,E2 -326.328} C_VEL
LIN {X 0,Y 608.444,Z 182.004,A -85,B 0,C 180,E1 -328.732,E2 -328.732} C_VEL
LIN {X 0,Y 608.474,Z 181.998,A -85,B 0,C 180,E1 -331.379,E2 -331.379} C_VEL
LIN {X 0,Y 608.469,Z 182.006,A -85,B 0,C 180,E1 -334.279,E2 -334.279} C_VEL
LIN {X 0,Y 608.449,Z 182.001,A -85,B 0,C 180,E1 -336.876,E2 -336.876} C_VEL
LIN {X 0,Y 608.462,Z 182.004,A -85,B 0,C 180,E1 -339.725,E2 -339.725} C_VEL
LIN {X 0,Y 608.444,Z 182.003,A -85,B 0,C 180,E1 -342.523,E2 -342.523} C_VEL
LIN {X 0,Y 608.471,Z 181.999,A -85,B 0,C 180,E1 -345.279,E2 -345.279} C_VEL
LIN {X 0,Y 608.457,Z 182.009,A -85,B 0,C 180,E1 -348,E2 -348} C_VEL
LIN {X 0,Y 608.458,Z 182,A -85,B 0,C 180,E1 -350.694,E2 -350.694} C_VEL
LIN {X 0,Y 608.474,Z 182.001,A -85,B 0,C 180,E1 -353.367,E2 -353.367} C_VEL
LIN {X 0,Y 608.444,Z 182.007,A -85,B 0,C 180,E1 -356.026,E2 -356.026} C_VEL
LIN {X 0,Y 608.456,Z 181.999,A -85,B 0,C 180,E1 -358.676,E2 -358.676} C_VEL
LIN {X 0,Y 608.471,Z 182.002,A -85,B 0,C 180,E1 -361.323,E2 -361.323} C_VEL
LIN {X 0,Y 608.441,Z 182.006,A -85,B 0,C 180,E1 -363.974,E2 -363.974} C_VEL
LIN {X 0,Y 608.454,Z 182,A -85,B 0,C 180,E1 -366.632,E2 -366.632} C_VEL
LIN {X 0,Y 608.47,Z 182.004,A -85,B 0,C 180,E1 -369.305,E2 -369.305} C_VEL
LIN {X 0,Y 608.446,Z 182.004,A -85,B 0,C 180,E1 -372,E2 -372} C_VEL
LIN {X 0,Y 608.466,Z 181.999,A -85,B 0,C 180,E1 -374.72,E2 -374.72} C_VEL
LIN {X 0,Y 608.449,Z 182.01,A -85,B 0,C 180,E1 -377.476,E2 -377.476} C_VEL
LIN {X 0,Y 608.44,Z 182.001,A -85,B 0,C 180,E1 -380.275,E2 -380.275} C_VEL
LIN {X 0,Y 608.454,Z 182,A -85,B 0,C 180,E1 -382.476,E2 -382.476} C_VEL
LIN {X 0,Y 608.445,Z 182.012,A -85,B 0,C 180,E1 -385.301,E2 -385.301} C_VEL
LIN {X 0,Y 608.437,Z 182.008,A -85,B 0,C 180,E1 -387.518,E2 -387.518} C_VEL
LIN {X 0,Y 608.438,Z 182.002,A -85,B 0,C 180,E1 -389.967,E2 -389.967} C_VEL
LIN {X 0,Y 608.455,Z 182.001,A -85,B 0,C 180,E1 -392.522,E2 -392.522} C_VEL
LIN {X 0,Y 608.428,Z 182.011,A -85,B 0,C 180,E1 -395.278,E2 -395.278} C_VEL
LIN {X 0,Y 608.448,Z 182.002,A -85,B 0,C 180,E1 -397.747,E2 -397.747} C_VEL
LIN {X 0,Y 608.439,Z 182.002,A -85,B 0,C 180,E1 -400.328,E2 -400.328} C_VEL
LIN {X 0,Y 608.46,Z 182.004,A -85,B 0,C 180,E1 -403.308,E2 -403.308} C_VEL
LIN {X 0,Y 608.447,Z 182.001,A -85,B 0,C 180,E1 -406.128,E2 -406.128} C_VEL
LIN {X 0,Y 608.457,Z 182.009,A -85,B 0,C 180,E1 -408.823,E2 -408.823} C_VEL
LIN {X 0,Y 608.421,Z 182.006,A -85,B 0,C 180,E1 -411.408,E2 -411.408} C_VEL
LIN {X 0,Y 608.438,Z 182.002,A -85,B 0,C 180,E1 -413.955,E2 -413.955} C_VEL
LIN {X 0,Y 608.467,Z 182.002,A -85,B 0,C 180,E1 -416.329,E2 -416.329} C_VEL
LIN {X 0,Y 608.445,Z 182.012,A -85,B 0,C 180,E1 -418.732,E2 -418.732} C_VEL
LIN {X 0,Y 608.436,Z 182.004,A -85,B 0,C 180,E1 -421.386,E2 -421.386} C_VEL
LIN {X 0,Y 608.458,Z 182.142,A -85,B 0,C 180,E1 -423.353,E2 -423.353} C_VEL
LIN {X 0,Y 608.799,Z 186.144,A -85,B 0,C 180,E1 -423.704,E2 -423.704} C_VEL
LIN {X 0,Y 608.749,Z 219.268,A -85,B 0,C 180,E1 -426.437,E2 -426.437} C_VEL
LIN {X 0,Y 608.705,Z 235.002,A -85,B 0,C 180,E1 -427.715,E2 -427.715} C_VEL
LIN {X 0,Y 608.907,Z 243.7,A -85,B 0,C 180,E1 -427.834,E2 -427.834} C_VEL
LIN {X 0,Y 608.804,Z 442.373,A -85,B 0,C 180,E1 -430.309,E2 -430.309} C_VEL
LIN {X 0,Y 608.795,Z 458.96,A -85,B 0,C 180,E1 -430.659,E2 -430.659} C_VEL
LIN {X 0,Y 608.744,Z 475.202,A -85,B 0,C 180,E1 -431.139,E2 -431.139} C_VEL
LIN {X 0,Y 608.688,Z 491.193,A -85,B 0,C 180,E1 -431.752,E2 -431.752} C_VEL
LIN {X 0,Y 608.681,Z 505.712,A -85,B 0,C 180,E1 -432.443,E2 -432.443} C_VEL
LIN {X 0,Y 608.633,Z 520.92,A -85,B 0,C 180,E1 -433.323,E2 -433.323} C_VEL
LIN {X 0,Y 608.574,Z 534.354,A -85,B 0,C 180,E1 -434.252,E2 -434.252} C_VEL
LIN {X 0,Y 608.548,Z 547.055,A -85,B 0,C 180,E1 -435.28,E2 -435.28} C_VEL
LIN {X 0,Y 608.496,Z 559.624,A -85,B 0,C 180,E1 -436.473,E2 -436.473} C_VEL
LIN {X 0,Y 608.47,Z 570.321,A -85,B 0,C 180,E1 -437.661,E2 -437.661} C_VEL
LIN {X 0,Y 608.474,Z 580.866,A -85,B 0,C 180,E1 -439.041,E2 -439.041} C_VEL
LIN {X 0,Y 608.466,Z 589.276,A -85,B 0,C 180,E1 -440.357,E2 -440.357} C_VEL
LIN {X 0,Y 608.452,Z 596.479,A -85,B 0,C 180,E1 -441.697,E2 -441.697} C_VEL
LIN {X 0,Y 608.438,Z 602.463,A -85,B 0,C 180,E1 -443.032,E2 -443.032} C_VEL
LIN {X 0,Y 608.435,Z 608.241,A -85,B 0,C 180,E1 -444.696,E2 -444.696} C_VEL
LIN {X 0,Y 608.43,Z 611.629,A -85,B 0,C 180,E1 -446.024,E2 -446.024} C_VEL
LIN {X 0,Y 608.412,Z 614.083,A -85,B 0,C 180,E1 -447.35,E2 -447.35} C_VEL
LIN {X 0,Y 608.441,Z 615.476,A -85,B 0,C 180,E1 -448.675,E2 -448.675} C_VEL
LIN {X 0,Y 608.429,Z 616,A -85,B 0,C 180,E1 -449.998,E2 -449.998} C_VEL
LIN {X 0,Y 608.44,Z 615.478,A -85,B 0,C 180,E1 -451.322,E2 -451.322} C_VEL
LIN {X 0,Y 608.412,Z 614.088,A -85,B 0,C 180,E1 -452.647,E2 -452.647} C_VEL
LIN {X 0,Y 608.43,Z 611.636,A -85,B 0,C 180,E1 -453.972,E2 -453.972} C_VEL
LIN {X 0,Y 608.435,Z 608.251,A -85,B 0,C 180,E1 -455.3,E2 -455.3} C_VEL
LIN {X 0,Y 608.436,Z 602.476,A -85,B 0,C 180,E1 -456.964,E2 -456.964} C_VEL
LIN {X 0,Y 608.443,Z 594.867,A -85,B 0,C 180,E1 -458.634,E2 -458.634} C_VEL
LIN {X 0,Y 608.461,Z 586.257,A -85,B 0,C 180,E1 -460.143,E2 -460.143} C_VEL
LIN {X 0,Y 608.466,Z 576.983,A -85,B 0,C 180,E1 -461.491,E2 -461.491} C_VEL
LIN {X 0,Y 608.49,Z 567.44,A -85,B 0,C 180,E1 -462.674,E2 -462.674} C_VEL
LIN {X 0,Y 608.524,Z 555.952,A -85,B 0,C 180,E1 -463.897,E2 -463.897} C_VEL
LIN {X 0,Y 608.552,Z 544.169,A -85,B 0,C 180,E1 -464.973,E2 -464.973} C_VEL
LIN {X 0,Y 608.597,Z 530.916,A -85,B 0,C 180,E1 -466.002,E2 -466.002} C_VEL
LIN {X 0,Y 608.616,Z 517.877,A -85,B 0,C 180,E1 -466.863,E2 -466.863} C_VEL
LIN {X 0,Y 608.677,Z 502.309,A -85,B 0,C 180,E1 -467.728,E2 -467.728} C_VEL
LIN {X 0,Y 608.711,Z 487.407,A -85,B 0,C 180,E1 -468.409,E2 -468.409} C_VEL
LIN {X 0,Y 608.736,Z 471.42,A -85,B 0,C 180,E1 -468.989,E2 -468.989} C_VEL
LIN {X 0,Y 608.792,Z 455.45,A -85,B 0,C 180,E1 -469.425,E2 -469.425} C_VEL
LIN {X 0,Y 608.807,Z 439.604,A -85,B 0,C 180,E1 -469.732,E2 -469.732} C_VEL
LIN {X 0,Y 608.91,Z 236.821,A -85,B 0,C 180,E1 -472.252,E2 -472.252} C_VEL
LIN {X 0,Y 608.719,Z 234.768,A -85,B 0,C 180,E1 -472.304,E2 -472.304} C_VEL
LIN {X 0,Y 608.772,Z 201.645,A -85,B 0,C 180,E1 -475.01,E2 -475.01} C_VEL
LIN {X 0,Y 608.807,Z 183.979,A -85,B 0,C 180,E1 -476.477,E2 -476.477} C_VEL
LIN {X 0,Y 608.415,Z 182.009,A -85,B 0,C 180,E1 -476.68,E2 -476.68} C_VEL
LIN {X 0,Y 608.465,Z 182.002,A -85,B 0,C 180,E1 -479.777,E2 -479.777} C_VEL
LIN {X 0,Y 608.419,Z 182.004,A -85,B 0,C 180,E1 -482.517,E2 -482.517} C_VEL
LIN {X 0,Y 608.448,Z 182.005,A -85,B 0,C 180,E1 -484.906,E2 -484.906} C_VEL
LIN {X 0,Y 608.448,Z 182.003,A -85,B 0,C 180,E1 -487.744,E2 -487.744} C_VEL
LIN {X 0,Y 608.41,Z 182.005,A -85,B 0,C 180,E1 -490.325,E2 -490.325} C_VEL
LIN {X 0,Y 608.437,Z 182.009,A -85,B 0,C 180,E1 -492.957,E2 -492.957} C_VEL
LIN {X 0,Y 608.43,Z 182.004,A -85,B 0,C 180,E1 -495.734,E2 -495.734} C_VEL
LIN {X 0,Y 608.431,Z 182.003,A -85,B 0,C 180,E1 -497.936,E2 -497.936} C_VEL
LIN {X 0,Y 608.453,Z 182.004,A -85,B 0,C 180,E1 -500.699,E2 -500.699} C_VEL
LIN {X 0,Y 608.455,Z 182.01,A -85,B 0,C 180,E1 -503.085,E2 -503.085} C_VEL
LIN {X 0,Y 608.461,Z 182.002,A -85,B 0,C 180,E1 -505.531,E2 -505.531} C_VEL
LIN {X 0,Y 608.435,Z 182.002,A -85,B 0,C 180,E1 -507.904,E2 -507.904} C_VEL
LIN {X 0,Y 608.42,Z 182.004,A -85,B 0,C 180,E1 -510.218,E2 -510.218} C_VEL
LIN {X 0,Y 608.47,Z 182.005,A -85,B 0,C 180,E1 -512.787,E2 -512.787} C_VEL
LIN {X 0,Y 608.436,Z 182.002,A -85,B 0,C 180,E1 -515.848,E2 -515.848} C_VEL
LIN {X 0,Y 608.434,Z 182.004,A -85,B 0,C 180,E1 -518.307,E2 -518.307} C_VEL
LIN {X 0,Y 608.45,Z 182.004,A -85,B 0,C 180,E1 -521.278,E2 -521.278} C_VEL
LIN {X 0,Y 608.419,Z 182.004,A -85,B 0,C 180,E1 -523.905,E2 -523.905} C_VEL
LIN {X 0,Y 608.455,Z 182.007,A -85,B 0,C 180,E1 -526.644,E2 -526.644} C_VEL
LIN {X 0,Y 608.445,Z 182.003,A -85,B 0,C 180,E1 -529.35,E2 -529.35} C_VEL
LIN {X 0,Y 608.432,Z 182.003,A -85,B 0,C 180,E1 -532.033,E2 -532.033} C_VEL
LIN {X 0,Y 608.467,Z 182.008,A -85,B 0,C 180,E1 -534.698,E2 -534.698} C_VEL
LIN {X 0,Y 608.449,Z 182.001,A -85,B 0,C 180,E1 -537.352,E2 -537.352} C_VEL
LIN {X 0,Y 608.429,Z 182.004,A -85,B 0,C 180,E1 -540,E2 -540} C_VEL
LIN {X 0,Y 608.473,Z 182.008,A -85,B 0,C 180,E1 -542.648,E2 -542.648} C_VEL
LIN {X 0,Y 608.438,Z 182.003,A -85,B 0,C 180,E1 -545.302,E2 -545.302} C_VEL
LIN {X 0,Y 608.452,Z 182.001,A -85,B 0,C 180,E1 -547.3,E2 -547.3} C_VEL
LIN {X 0,Y 608.425,Z 182.003,A -85,B 0,C 180,E1 -549.49,E2 -549.49} C_VEL
LIN {X 0,Y 607.739,Z 182.092,A -85,B 0,C 180,E1 -550.043,E2 -550.043} C_VEL
LIN {X 0,Y 604.879,Z 182.449,A -85,B 0,C 180,E1 -550.94,E2 -550.94} C_VEL
LIN {X 0,Y 602.481,Z 182.747,A -85,B 0,C 180,E1 -551.662,E2 -551.662} C_VEL
LIN {X 0,Y 601.462,Z 182.874,A -85,B 0,C 180,E1 -552.218,E2 -552.218} C_VEL
LIN {X 0,Y 601.384,Z 182.883,A -85,B 0,C 180,E1 -552.407,E2 -552.407} C_VEL
LIN {X 0,Y 601.41,Z 182.882,A -85,B 0,C 180,E1 -554.898,E2 -554.898} C_VEL
LIN {X 0,Y 601.406,Z 182.88,A -85,B 0,C 180,E1 -556.987,E2 -556.987} C_VEL
LIN {X 0,Y 601.374,Z 182.882,A -85,B 0,C 180,E1 -559.811,E2 -559.811} C_VEL
LIN {X 0,Y 601.392,Z 182.882,A -85,B 0,C 180,E1 -561.96,E2 -561.96} C_VEL
LIN {X 0,Y 601.409,Z 182.885,A -85,B 0,C 180,E1 -564.296,E2 -564.296} C_VEL
LIN {X 0,Y 601.42,Z 182.876,A -85,B 0,C 180,E1 -567.113,E2 -567.113} C_VEL
LIN {X 0,Y 601.386,Z 182.88,A -85,B 0,C 180,E1 -569.395,E2 -569.395} C_VEL
LIN {X 0,Y 601.378,Z 182.882,A -85,B 0,C 180,E1 -571.729,E2 -571.729} C_VEL
LIN {X 0,Y 601.399,Z 182.885,A -85,B 0,C 180,E1 -574.121,E2 -574.121} C_VEL
LIN {X 0,Y 601.387,Z 182.886,A -85,B 0,C 180,E1 -576.585,E2 -576.585} C_VEL
LIN {X 0,Y 601.377,Z 182.881,A -85,B 0,C 180,E1 -579.13,E2 -579.13} C_VEL
LIN {X 0,Y 601.401,Z 182.881,A -85,B 0,C 180,E1 -581.768,E2 -581.768} C_VEL
LIN {X 0,Y 601.405,Z 182.882,A -85,B 0,C 180,E1 -584.538,E2 -584.538} C_VEL
LIN {X 0,Y 601.359,Z 182.884,A -85,B 0,C 180,E1 -587.329,E2 -587.329} C_VEL
LIN {X 0,Y 601.386,Z 182.888,A -85,B 0,C 180,E1 -590.007,E2 -590.007} C_VEL
LIN {X 0,Y 601.416,Z 182.879,A -85,B 0,C 180,E1 -592.621,E2 -592.621} C_VEL
LIN {X 0,Y 601.372,Z 182.881,A -85,B 0,C 180,E1 -595.069,E2 -595.069} C_VEL
LIN {X 0,Y 601.392,Z 182.881,A -85,B 0,C 180,E1 -597.485,E2 -597.485} C_VEL
LIN {X 0,Y 601.419,Z 182.883,A -85,B 0,C 180,E1 -599.854,E2 -599.854} C_VEL
LIN {X 0,Y 601.395,Z 182.879,A -85,B 0,C 180,E1 -602.889,E2 -602.889} C_VEL
LIN {X 0,Y 601.41,Z 182.883,A -85,B 0,C 180,E1 -605.714,E2 -605.714} C_VEL
LIN {X 0,Y 601.387,Z 182.89,A -85,B 0,C 180,E1 -608.042,E2 -608.042} C_VEL
LIN {X 0,Y 601.398,Z 182.878,A -85,B 0,C 180,E1 -610.903,E2 -610.903} C_VEL
LIN {X 0,Y 601.411,Z 182.884,A -85,B 0,C 180,E1 -613.715,E2 -613.715} C_VEL
LIN {X 0,Y 601.395,Z 182.881,A -85,B 0,C 180,E1 -616.486,E2 -616.486} C_VEL
LIN {X 0,Y 601.368,Z 182.884,A -85,B 0,C 180,E1 -619.225,E2 -619.225} C_VEL
LIN {X 0,Y 601.433,Z 182.884,A -85,B 0,C 180,E1 -621.941,E2 -621.941} C_VEL
LIN {X 0,Y 601.391,Z 182.88,A -85,B 0,C 180,E1 -624.637,E2 -624.637} C_VEL
LIN {X 0,Y 601.41,Z 182.881,A -85,B 0,C 180,E1 -627.323,E2 -627.323} C_VEL
LIN {X 0,Y 601.446,Z 182.881,A -85,B 0,C 180,E1 -630.002,E2 -630.002} C_VEL
LIN {X 0,Y 601.419,Z 183.076,A -85,B 0,C 180,E1 -632.346,E2 -632.346} C_VEL
LIN {X 0,Y 601.909,Z 186.371,A -85,B 0,C 180,E1 -632.678,E2 -632.678} C_VEL
LIN {X 0,Y 601.857,Z 205.837,A -85,B 0,C 180,E1 -634.501,E2 -634.501} C_VEL
LIN {X 0,Y 602.318,Z 208.738,A -85,B 0,C 180,E1 -634.561,E2 -634.561} C_VEL
LIN {X 0,Y 602.131,Z 412.143,A -85,B 0,C 180,E1 -637.123,E2 -637.123} C_VEL
LIN {X 0,Y 602.082,Z 429.18,A -85,B 0,C 180,E1 -637.484,E2 -637.484} C_VEL
LIN {X 0,Y 602.007,Z 445.394,A -85,B 0,C 180,E1 -637.97,E2 -637.97} C_VEL
LIN {X 0,Y 601.911,Z 460.724,A -85,B 0,C 180,E1 -638.563,E2 -638.563} C_VEL
LIN {X 0,Y 601.833,Z 476.536,A -85,B 0,C 180,E1 -639.326,E2 -639.326} C_VEL
LIN {X 0,Y 601.755,Z 490.979,A -85,B 0,C 180,E1 -640.176,E2 -640.176} C_VEL
LIN {X 0,Y 601.673,Z 504.605,A -85,B 0,C 180,E1 -641.13,E2 -641.13} C_VEL
LIN {X 0,Y 601.572,Z 516.948,A -85,B 0,C 180,E1 -642.14,E2 -642.14} C_VEL
LIN {X 0,Y 601.505,Z 529.49,A -85,B 0,C 180,E1 -643.343,E2 -643.343} C_VEL
LIN {X 0,Y 601.462,Z 540.259,A -85,B 0,C 180,E1 -644.551,E2 -644.551} C_VEL
LIN {X 0,Y 601.414,Z 550.758,A -85,B 0,C 180,E1 -645.94,E2 -645.94} C_VEL
LIN {X 0,Y 601.397,Z 559.581,A -85,B 0,C 180,E1 -647.338,E2 -647.338} C_VEL
LIN {X 0,Y 601.379,Z 567.261,A -85,B 0,C 180,E1 -648.807,E2 -648.807} C_VEL
LIN {X 0,Y 601.369,Z 573.11,A -85,B 0,C 180,E1 -650.168,E2 -650.168} C_VEL
LIN {X 0,Y 601.342,Z 578.001,A -85,B 0,C 180,E1 -651.602,E2 -651.602} C_VEL
LIN {X 0,Y 601.328,Z 580.913,A -85,B 0,C 180,E1 -652.687,E2 -652.687} C_VEL
LIN {X 0,Y 601.312,Z 583.921,A -85,B 0,C 180,E1 -654.265,E2 -654.265} C_VEL
LIN {X 0,Y 601.337,Z 585.579,A -85,B 0,C 180,E1 -655.851,E2 -655.851} C_VEL
LIN {X 0,Y 601.352,Z 585.935,A -85,B 0,C 180,E1 -657.35,E2 -657.35} C_VEL
LIN {X 0,Y 601.33,Z 585.207,A -85,B 0,C 180,E1 -658.769,E2 -658.769} C_VEL
LIN {X 0,Y 601.346,Z 583.354,A -85,B 0,C 180,E1 -660.169,E2 -660.169} C_VEL
LIN {X 0,Y 601.342,Z 580.074,A -85,B 0,C 180,E1 -661.731,E2 -661.731} C_VEL
LIN {X 0,Y 601.368,Z 575.331,A -85,B 0,C 180,E1 -663.318,E2 -663.318} C_VEL
LIN {X 0,Y 601.343,Z 570.636,A -85,B 0,C 180,E1 -664.53,E2 -664.53} C_VEL
LIN {X 0,Y 601.384,Z 563.678,A -85,B 0,C 180,E1 -666.005,E2 -666.005} C_VEL
LIN {X 0,Y 601.418,Z 555.562,A -85,B 0,C 180,E1 -667.421,E2 -667.421} C_VEL
LIN {X 0,Y 601.425,Z 546.29,A -85,B 0,C 180,E1 -668.768,E2 -668.768} C_VEL
LIN {X 0,Y 601.463,Z 536.397,A -85,B 0,C 180,E1 -669.991,E2 -669.991} C_VEL
LIN {X 0,Y 601.52,Z 525.021,A -85,B 0,C 180,E1 -671.199,E2 -671.199} C_VEL
LIN {X 0,Y 601.632,Z 512.878,A -85,B 0,C 180,E1 -672.301,E2 -672.301} C_VEL
LIN {X 0,Y 601.703,Z 499.611,A -85,B 0,C 180,E1 -673.331,E2 -673.331} C_VEL
LIN {X 0,Y 601.791,Z 485.565,A -85,B 0,C 180,E1 -674.25,E2 -674.25} C_VEL
LIN {X 0,Y 601.877,Z 471.343,A -85,B 0,C 180,E1 -675.029,E2 -675.029} C_VEL
LIN {X 0,Y 601.967,Z 456.653,A -85,B 0,C 180,E1 -675.699,E2 -675.699} C_VEL
LIN {X 0,Y 602.023,Z 439.996,A -85,B 0,C 180,E1 -676.3,E2 -676.3} C_VEL
LIN {X 0,Y 602.103,Z 423.511,A -85,B 0,C 180,E1 -676.743,E2 -676.743} C_VEL
LIN {X 0,Y 602.132,Z 406.439,A -85,B 0,C 180,E1 -677.053,E2 -677.053} C_VEL
LIN {X 0,Y 602.325,Z 208.176,A -85,B 0,C 180,E1 -679.536,E2 -679.536} C_VEL
LIN {X 0,Y 601.885,Z 205.753,A -85,B 0,C 180,E1 -679.595,E2 -679.595} C_VEL
LIN {X 0,Y 601.988,Z 185.797,A -85,B 0,C 180,E1 -681.462,E2 -681.462} C_VEL
LIN {X 0,Y 601.419,Z 182.883,A -85,B 0,C 180,E1 -681.785,E2 -681.785} C_VEL
LIN {X 0,Y 601.399,Z 182.889,A -85,B 0,C 180,E1 -684.246,E2 -684.246} C_VEL
LIN {X 0,Y 601.418,Z 182.881,A -85,B 0,C 180,E1 -686.685,E2 -686.685} C_VEL
LIN {X 0,Y 601.411,Z 182.878,A -85,B 0,C 180,E1 -689.057,E2 -689.057} C_VEL
LIN {X 0,Y 601.433,Z 182.875,A -85,B 0,C 180,E1 -691.373,E2 -691.373} C_VEL
LIN {X 0,Y 601.411,Z 182.888,A -85,B 0,C 180,E1 -694.132,E2 -694.132} C_VEL
LIN {X 0,Y 601.417,Z 182.879,A -85,B 0,C 180,E1 -696.589,E2 -696.589} C_VEL
LIN {X 0,Y 601.431,Z 182.876,A -85,B 0,C 180,E1 -699.478,E2 -699.478} C_VEL
LIN {X 0,Y 601.393,Z 182.884,A -85,B 0,C 180,E1 -702.311,E2 -702.311} C_VEL
LIN {X 0,Y 601.408,Z 182.881,A -85,B 0,C 180,E1 -704.408,E2 -704.408} C_VEL
LIN {X 0,Y 601.416,Z 182.877,A -85,B 0,C 180,E1 -707.171,E2 -707.171} C_VEL
LIN {X 0,Y 601.426,Z 182.886,A -85,B 0,C 180,E1 -709.904,E2 -709.904} C_VEL
LIN {X 0,Y 601.433,Z 182.875,A -85,B 0,C 180,E1 -712.614,E2 -712.614} C_VEL
LIN {X 0,Y 601.421,Z 182.879,A -85,B 0,C 180,E1 -715.308,E2 -715.308} C_VEL
LIN {X 0,Y 601.414,Z 182.883,A -85,B 0,C 180,E1 -717.991,E2 -717.991} C_VEL
LIN {X 0,Y 601.439,Z 182.874,A -85,B 0,C 180,E1 -720.669,E2 -720.669} C_VEL
LIN {X 0,Y 601.431,Z 182.88,A -85,B 0,C 180,E1 -723.349,E2 -723.349} C_VEL
LIN {X 0,Y 601.399,Z 182.882,A -85,B 0,C 180,E1 -726.037,E2 -726.037} C_VEL
LIN {X 0,Y 601.428,Z 182.878,A -85,B 0,C 180,E1 -728.061,E2 -728.061} C_VEL
LIN {X 0,Y 601.421,Z 182.878,A -85,B 0,C 180,E1 -731.013,E2 -731.013} C_VEL
LIN {X 0,Y 601.409,Z 182.888,A -85,B 0,C 180,E1 -733.516,E2 -733.516} C_VEL
LIN {X 0,Y 601.421,Z 182.876,A -85,B 0,C 180,E1 -736.287,E2 -736.287} C_VEL
LIN {X 0,Y 601.413,Z 182.882,A -85,B 0,C 180,E1 -739.099,E2 -739.099} C_VEL
LIN {X 0,Y 601.405,Z 182.886,A -85,B 0,C 180,E1 -741.239,E2 -741.239} C_VEL
LIN {X 0,Y 601.433,Z 182.875,A -85,B 0,C 180,E1 -744.141,E2 -744.141} C_VEL
LIN {X 0,Y 601.452,Z 182.88,A -85,B 0,C 180,E1 -747.111,E2 -747.111} C_VEL
LIN {X 0,Y 601.404,Z 182.886,A -85,B 0,C 180,E1 -749.394,E2 -749.394} C_VEL
LIN {X 0,Y 601.396,Z 182.881,A -85,B 0,C 180,E1 -751.727,E2 -751.727} C_VEL
LIN {X 0,Y 601.416,Z 182.876,A -85,B 0,C 180,E1 -754.119,E2 -754.119} C_VEL
LIN {X 0,Y 601.433,Z 182.88,A -85,B 0,C 180,E1 -757.382,E2 -757.382} C_VEL
LIN {X 0,Y 601.396,Z 182.879,A -85,B 0,C 180,E1 -759.996,E2 -759.996} C_VEL
LIN {X 0,Y 601.409,Z 182.882,A -85,B 0,C 180,E1 -762.67,E2 -762.67} C_VEL
LIN {X 0,Y 601.397,Z 182.882,A -85,B 0,C 180,E1 -765.479,E2 -765.479} C_VEL
LIN {X 0,Y 601.419,Z 182.879,A -85,B 0,C 180,E1 -768.407,E2 -768.407} C_VEL
LIN {X 0,Y 601.426,Z 182.886,A -85,B 0,C 180,E1 -770.874,E2 -770.874} C_VEL
LIN {X 0,Y 601.392,Z 182.882,A -85,B 0,C 180,E1 -773.416,E2 -773.416} C_VEL
LIN {X 0,Y 601.428,Z 182.876,A -85,B 0,C 180,E1 -776.065,E2 -776.065} C_VEL
LIN {X 0,Y 601.396,Z 182.885,A -85,B 0,C 180,E1 -779.056,E2 -779.056} C_VEL
LIN {X 0,Y 601.397,Z 182.882,A -85,B 0,C 180,E1 -781.371,E2 -781.371} C_VEL
LIN {X 0,Y 601.424,Z 182.97,A -85,B 0,C 180,E1 -783.086,E2 -783.086} C_VEL
LIN {X 0,Y 602.156,Z 187.249,A -85,B 0,C 180,E1 -783.484,E2 -783.484} C_VEL
LIN {X 0,Y 602.047,Z 218.164,A -85,B 0,C 180,E1 -786.067,E2 -786.067} C_VEL
LIN {X 0,Y 602.023,Z 235.337,A -85,B 0,C 180,E1 -787.461,E2 -787.461} C_VEL
LIN {X 0,Y 602.356,Z 238.908,A -85,B 0,C 180,E1 -787.519,E2 -787.519} C_VEL
LIN {X 0,Y 602.122,Z 442.373,A -85,B 0,C 180,E1 -790.081,E2 -790.081} C_VEL
LIN {X 0,Y 602.083,Z 458.961,A -85,B 0,C 180,E1 -790.435,E2 -790.435} C_VEL
LIN {X 0,Y 602.013,Z 473.912,A -85,B 0,C 180,E1 -790.876,E2 -790.876} C_VEL
LIN {X 0,Y 601.916,Z 489.224,A -85,B 0,C 180,E1 -791.452,E2 -791.452} C_VEL
LIN {X 0,Y 601.869,Z 503.993,A -85,B 0,C 180,E1 -792.149,E2 -792.149} C_VEL
LIN {X 0,Y 601.756,Z 517.827,A -85,B 0,C 180,E1 -792.935,E2 -792.935} C_VEL
LIN {X 0,Y 601.696,Z 532.036,A -85,B 0,C 180,E1 -793.893,E2 -793.893} C_VEL
LIN {X 0,Y 601.593,Z 545.114,A -85,B 0,C 180,E1 -794.933,E2 -794.933} C_VEL
LIN {X 0,Y 601.556,Z 557.671,A -85,B 0,C 180,E1 -796.107,E2 -796.107} C_VEL
LIN {X 0,Y 601.472,Z 568.901,A -85,B 0,C 180,E1 -797.343,E2 -797.343} C_VEL
LIN {X 0,Y 601.428,Z 579.28,A -85,B 0,C 180,E1 -798.69,E2 -798.69} C_VEL
LIN {X 0,Y 601.388,Z 588.264,A -85,B 0,C 180,E1 -800.073,E2 -800.073} C_VEL
LIN {X 0,Y 601.365,Z 596.48,A -85,B 0,C 180,E1 -801.599,E2 -801.599} C_VEL
LIN {X 0,Y 601.363,Z 602.463,A -85,B 0,C 180,E1 -802.95,E2 -802.95} C_VEL
LIN {X 0,Y 601.346,Z 608.241,A -85,B 0,C 180,E1 -804.634,E2 -804.634} C_VEL
LIN {X 0,Y 601.339,Z 611.63,A -85,B 0,C 180,E1 -805.977,E2 -805.977} C_VEL
LIN {X 0,Y 601.311,Z 614.084,A -85,B 0,C 180,E1 -807.319,E2 -807.319} C_VEL
LIN {X 0,Y 601.341,Z 615.476,A -85,B 0,C 180,E1 -808.659,E2 -808.659} C_VEL
LIN {X 0,Y 601.33,Z 616,A -85,B 0,C 180,E1 -809.998,E2 -809.998} C_VEL
LIN {X 0,Y 601.34,Z 615.479,A -85,B 0,C 180,E1 -811.338,E2 -811.338} C_VEL
LIN {X 0,Y 601.311,Z 614.089,A -85,B 0,C 180,E1 -812.678,E2 -812.678} C_VEL
LIN {X 0,Y 601.339,Z 611.637,A -85,B 0,C 180,E1 -814.019,E2 -814.019} C_VEL
LIN {X 0,Y 601.346,Z 608.252,A -85,B 0,C 180,E1 -815.363,E2 -815.363} C_VEL
LIN {X 0,Y 601.363,Z 602.476,A -85,B 0,C 180,E1 -817.047,E2 -817.047} C_VEL
LIN {X 0,Y 601.376,Z 594.867,A -85,B 0,C 180,E1 -818.737,E2 -818.737} C_VEL
LIN {X 0,Y 601.41,Z 586.258,A -85,B 0,C 180,E1 -820.263,E2 -820.263} C_VEL
LIN {X 0,Y 601.428,Z 576.984,A -85,B 0,C 180,E1 -821.627,E2 -821.627} C_VEL
LIN {X 0,Y 601.479,Z 567.441,A -85,B 0,C 180,E1 -822.825,E2 -822.825} C_VEL
LIN {X 0,Y 601.54,Z 556.635,A -85,B 0,C 180,E1 -823.996,E2 -823.996} C_VEL
LIN {X 0,Y 601.601,Z 544.17,A -85,B 0,C 180,E1 -825.15,E2 -825.15} C_VEL
LIN {X 0,Y 601.706,Z 530.916,A -85,B 0,C 180,E1 -826.19,E2 -826.19} C_VEL
LIN {X 0,Y 601.784,Z 516.47,A -85,B 0,C 180,E1 -827.148,E2 -827.148} C_VEL
LIN {X 0,Y 601.862,Z 502.312,A -85,B 0,C 180,E1 -827.935,E2 -827.935} C_VEL
LIN {X 0,Y 601.941,Z 487.942,A -85,B 0,C 180,E1 -828.603,E2 -828.603} C_VEL
LIN {X 0,Y 602.007,Z 471.419,A -85,B 0,C 180,E1 -829.21,E2 -829.21} C_VEL
LIN {X 0,Y 602.087,Z 455.452,A -85,B 0,C 180,E1 -829.65,E2 -829.65} C_VEL
LIN {X 0,Y 602.143,Z 439.604,A -85,B 0,C 180,E1 -829.959,E2 -829.959} C_VEL
LIN {X 0,Y 602.313,Z 237.194,A -85,B 0,C 180,E1 -832.504,E2 -832.504} C_VEL
LIN {X 0,Y 601.94,Z 234.83,A -85,B 0,C 180,E1 -832.564,E2 -832.564} C_VEL
LIN {X 0,Y 602.068,Z 203.853,A -85,B 0,C 180,E1 -835.123,E2 -835.123} C_VEL
LIN {X 0,Y 602.164,Z 186.187,A -85,B 0,C 180,E1 -836.605,E2 -836.605} C_VEL
LIN {X 0,Y 601.396,Z 182.887,A -85,B 0,C 180,E1 -836.923,E2 -836.923} C_VEL
LIN {X 0,Y 601.396,Z 182.889,A -85,B 0,C 180,E1 -839.391,E2 -839.391} C_VEL
LIN {X 0,Y 601.393,Z 182.883,A -85,B 0,C 180,E1 -841.724,E2 -841.724} C_VEL
LIN {X 0,Y 601.408,Z 182.878,A -85,B 0,C 180,E1 -844.116,E2 -844.116} C_VEL
LIN {X 0,Y 601.38,Z 182.882,A -85,B 0,C 180,E1 -846.581,E2 -846.581} C_VEL
LIN {X 0,Y 601.425,Z 182.88,A -85,B 0,C 180,E1 -849.534,E2 -849.534} C_VEL
LIN {X 0,Y 601.4,Z 182.88,A -85,B 0,C 180,E1 -851.763,E2 -851.763} C_VEL
LIN {X 0,Y 601.427,Z 182.879,A -85,B 0,C 180,E1 -853.582,E2 -853.582} C_VEL
LIN {X 0,Y 601.402,Z 182.879,A -85,B 0,C 180,E1 -856.425,E2 -856.425} C_VEL
LIN {X 0,Y 601.41,Z 182.882,A -85,B 0,C 180,E1 -859.422,E2 -859.422} C_VEL
LIN {X 0,Y 601.393,Z 182.881,A -85,B 0,C 180,E1 -861.73,E2 -861.73} C_VEL
LIN {X 0,Y 601.359,Z 182.883,A -85,B 0,C 180,E1 -864.244,E2 -864.244} C_VEL
LIN {X 0,Y 601.389,Z 182.884,A -85,B 0,C 180,E1 -866.684,E2 -866.684} C_VEL
LIN {X 0,Y 601.406,Z 182.888,A -85,B 0,C 180,E1 -869.058,E2 -869.058} C_VEL
LIN {X 0,Y 601.42,Z 182.88,A -85,B 0,C 180,E1 -871.373,E2 -871.373} C_VEL
LIN {X 0,Y 601.378,Z 182.881,A -85,B 0,C 180,E1 -873.635,E2 -873.635} C_VEL
LIN {X 0,Y 601.394,Z 182.884,A -85,B 0,C 180,E1 -876.589,E2 -876.589} C_VEL
LIN {X 0,Y 601.408,Z 182.878,A -85,B 0,C 180,E1 -879.478,E2 -879.478} C_VEL
LIN {X 0,Y 601.39,Z 182.88,A -85,B 0,C 180,E1 -881.608,E2 -881.608} C_VEL
LIN {X 0,Y 601.393,Z 182.883,A -85,B 0,C 180,E1 -884.409,E2 -884.409} C_VEL
LIN {X 0,Y 601.403,Z 182.881,A -85,B 0,C 180,E1 -887.172,E2 -887.172} C_VEL
LIN {X 0,Y 601.411,Z 182.88,A -85,B 0,C 180,E1 -889.224,E2 -889.224} C_VEL
LIN {X 0,Y 601.399,Z 182.879,A -85,B 0,C 180,E1 -891.939,E2 -891.939} C_VEL
LIN {X 0,Y 601.424,Z 182.884,A -85,B 0,C 180,E1 -894.636,E2 -894.636} C_VEL
LIN {X 0,Y 601.415,Z 182.877,A -85,B 0,C 180,E1 -897.321,E2 -897.321} C_VEL
LIN {X 0,Y 601.398,Z 182.879,A -85,B 0,C 180,E1 -900,E2 -900} C_VEL
LIN {X 0,Y 601.435,Z 182.884,A -85,B 0,C 180,E1 -902.679,E2 -902.679} C_VEL
LIN {X 0,Y 601.399,Z 182.879,A -85,B 0,C 180,E1 -905.365,E2 -905.365} C_VEL
LIN {X 0,Y 601.403,Z 182.88,A -85,B 0,C 180,E1 -908.062,E2 -908.062} C_VEL
LIN {X 0,Y 601.411,Z 182.879,A -85,B 0,C 180,E1 -911.025,E2 -911.025} C_VEL
LIN {X 0,Y 601.384,Z 182.883,A -85,B 0,C 180,E1 -912.407,E2 -912.407} C_VEL
LIN {X 0,Y 600.73,Z 182.967,A -85,B 0,C 180,E1 -912.966,E2 -912.966} C_VEL
LIN {X 0,Y 597.88,Z 183.321,A -85,B 0,C 180,E1 -913.874,E2 -913.874} C_VEL
LIN {X 0,Y 595.462,Z 183.628,A -85,B 0,C 180,E1 -914.604,E2 -914.604} C_VEL
LIN {X 0,Y 594.42,Z 183.75,A -85,B 0,C 180,E1 -915.168,E2 -915.168} C_VEL
LIN {X 0,Y 594.334,Z 183.759,A -85,B 0,C 180,E1 -915.359,E2 -915.359} C_VEL
LIN {X 0,Y 594.36,Z 183.756,A -85,B 0,C 180,E1 -917.195,E2 -917.195} C_VEL
LIN {X 0,Y 594.344,Z 183.756,A -85,B 0,C 180,E1 -919.336,E2 -919.336} C_VEL
LIN {X 0,Y 594.341,Z 183.758,A -85,B 0,C 180,E1 -921.505,E2 -921.505} C_VEL
LIN {X 0,Y 594.36,Z 183.756,A -85,B 0,C 180,E1 -923.706,E2 -923.706} C_VEL
LIN {X 0,Y 594.359,Z 183.76,A -85,B 0,C 180,E1 -926.701,E2 -926.701} C_VEL
LIN {X 0,Y 594.362,Z 183.757,A -85,B 0,C 180,E1 -929,E2 -929} C_VEL
LIN {X 0,Y 594.351,Z 183.757,A -85,B 0,C 180,E1 -931.645,E2 -931.645} C_VEL
LIN {X 0,Y 594.356,Z 183.762,A -85,B 0,C 180,E1 -934.582,E2 -934.582} C_VEL
LIN {X 0,Y 594.359,Z 183.756,A -85,B 0,C 180,E1 -937.089,E2 -937.089} C_VEL
LIN {X 0,Y 594.332,Z 183.76,A -85,B 0,C 180,E1 -939.774,E2 -939.774} C_VEL
LIN {X 0,Y 594.373,Z 183.762,A -85,B 0,C 180,E1 -942.376,E2 -942.376} C_VEL
LIN {X 0,Y 594.324,Z 183.759,A -85,B 0,C 180,E1 -945.196,E2 -945.196} C_VEL
LIN {X 0,Y 594.362,Z 183.765,A -85,B 0,C 180,E1 -948.155,E2 -948.155} C_VEL
LIN {X 0,Y 594.352,Z 183.756,A -85,B 0,C 180,E1 -951.3,E2 -951.3} C_VEL
LIN {X 0,Y 594.354,Z 183.76,A -85,B 0,C 180,E1 -953.759,E2 -953.759} C_VEL
LIN {X 0,Y 594.366,Z 183.763,A -85,B 0,C 180,E1 -956.241,E2 -956.241} C_VEL
LIN {X 0,Y 594.352,Z 183.758,A -85,B 0,C 180,E1 -958.652,E2 -958.652} C_VEL
LIN {X 0,Y 594.363,Z 183.755,A -85,B 0,C 180,E1 -961.047,E2 -961.047} C_VEL
LIN {X 0,Y 594.349,Z 183.757,A -85,B 0,C 180,E1 -963.302,E2 -963.302} C_VEL
LIN {X 0,Y 594.351,Z 183.76,A -85,B 0,C 180,E1 -965.576,E2 -965.576} C_VEL
LIN {X 0,Y 594.344,Z 183.76,A -85,B 0,C 180,E1 -968.498,E2 -968.498} C_VEL
LIN {X 0,Y 594.349,Z 183.759,A -85,B 0,C 180,E1 -971.384,E2 -971.384} C_VEL
LIN {X 0,Y 594.343,Z 183.763,A -85,B 0,C 180,E1 -974.221,E2 -974.221} C_VEL
LIN {X 0,Y 594.366,Z 183.759,A -85,B 0,C 180,E1 -976.323,E2 -976.323} C_VEL
LIN {X 0,Y 594.344,Z 183.758,A -85,B 0,C 180,E1 -979.096,E2 -979.096} C_VEL
LIN {X 0,Y 594.377,Z 183.764,A -85,B 0,C 180,E1 -981.845,E2 -981.845} C_VEL
LIN {X 0,Y 594.361,Z 183.756,A -85,B 0,C 180,E1 -984.574,E2 -984.574} C_VEL
LIN {X 0,Y 594.377,Z 183.757,A -85,B 0,C 180,E1 -987.291,E2 -987.291} C_VEL
LIN {X 0,Y 594.414,Z 183.757,A -85,B 0,C 180,E1 -990.002,E2 -990.002} C_VEL
LIN {X 0,Y 594.4,Z 183.962,A -85,B 0,C 180,E1 -992.119,E2 -992.119} C_VEL
LIN {X 0,Y 595.153,Z 188.003,A -85,B 0,C 180,E1 -992.54,E2 -992.54} C_VEL
LIN {X 0,Y 595.061,Z 205.894,A -85,B 0,C 180,E1 -994.235,E2 -994.235} C_VEL
LIN {X 0,Y 595.766,Z 209.889,A -85,B 0,C 180,E1 -994.314,E2 -994.314} C_VEL
LIN {X 0,Y 595.468,Z 411.812,A -85,B 0,C 180,E1 -996.886,E2 -996.886} C_VEL
LIN {X 0,Y 595.389,Z 429.14,A -85,B 0,C 180,E1 -997.253,E2 -997.253} C_VEL
LIN {X 0,Y 595.272,Z 444.65,A -85,B 0,C 180,E1 -997.719,E2 -997.719} C_VEL
LIN {X 0,Y 595.17,Z 460.134,A -85,B 0,C 180,E1 -998.318,E2 -998.318} C_VEL
LIN {X 0,Y 595.028,Z 476.063,A -85,B 0,C 180,E1 -999.091,E2 -999.091} C_VEL
LIN {X 0,Y 594.879,Z 490.6,A -85,B 0,C 180,E1 -999.951,E2 -999.951} C_VEL
LIN {X 0,Y 594.772,Z 505.085,A -85,B 0,C 180,E1 -1000.976,E2 -1000.976} C_VEL
LIN {X 0,Y 594.606,Z 518.612,A -85,B 0,C 180,E1 -1002.112,E2 -1002.112} C_VEL
LIN {X 0,Y 594.495,Z 530.904,A -85,B 0,C 180,E1 -1003.329,E2 -1003.329} C_VEL
LIN {X 0,Y 594.436,Z 541.447,A -85,B 0,C 180,E1 -1004.552,E2 -1004.552} C_VEL
LIN {X 0,Y 594.372,Z 550.579,A -85,B 0,C 180,E1 -1005.782,E2 -1005.782} C_VEL
LIN {X 0,Y 594.326,Z 559.435,A -85,B 0,C 180,E1 -1007.196,E2 -1007.196} C_VEL
LIN {X 0,Y 594.291,Z 566.857,A -85,B 0,C 180,E1 -1008.621,E2 -1008.621} C_VEL
LIN {X 0,Y 594.268,Z 573.014,A -85,B 0,C 180,E1 -1010.058,E2 -1010.058} C_VEL
LIN {X 0,Y 594.247,Z 577.914,A -85,B 0,C 180,E1 -1011.509,E2 -1011.509} C_VEL
LIN {X 0,Y 594.216,Z 581.63,A -85,B 0,C 180,E1 -1012.974,E2 -1012.974} C_VEL
LIN {X 0,Y 594.213,Z 584.246,A -85,B 0,C 180,E1 -1014.455,E2 -1014.455} C_VEL
LIN {X 0,Y 594.228,Z 585.685,A -85,B 0,C 180,E1 -1015.99,E2 -1015.99} C_VEL
LIN {X 0,Y 594.257,Z 585.901,A -85,B 0,C 180,E1 -1017.502,E2 -1017.502} C_VEL
LIN {X 0,Y 594.251,Z 584.973,A -85,B 0,C 180,E1 -1019.006,E2 -1019.006} C_VEL
LIN {X 0,Y 594.231,Z 582.765,A -85,B 0,C 180,E1 -1020.569,E2 -1020.569} C_VEL
LIN {X 0,Y 594.231,Z 579.112,A -85,B 0,C 180,E1 -1022.156,E2 -1022.156} C_VEL
LIN {X 0,Y 594.273,Z 573.969,A -85,B 0,C 180,E1 -1023.768,E2 -1023.768} C_VEL
LIN {X 0,Y 594.306,Z 567.574,A -85,B 0,C 180,E1 -1025.316,E2 -1025.316} C_VEL
LIN {X 0,Y 594.319,Z 560.235,A -85,B 0,C 180,E1 -1026.756,E2 -1026.756} C_VEL
LIN {X 0,Y 594.372,Z 551.754,A -85,B 0,C 180,E1 -1028.132,E2 -1028.132} C_VEL
LIN {X 0,Y 594.441,Z 542.092,A -85,B 0,C 180,E1 -1029.456,E2 -1029.456} C_VEL
LIN {X 0,Y 594.533,Z 531.495,A -85,B 0,C 180,E1 -1030.697,E2 -1030.697} C_VEL
LIN {X 0,Y 594.618,Z 519.176,A -85,B 0,C 180,E1 -1031.927,E2 -1031.927} C_VEL
LIN {X 0,Y 594.75,Z 506.368,A -85,B 0,C 180,E1 -1033.015,E2 -1033.015} C_VEL
LIN {X 0,Y 594.871,Z 493.109,A -85,B 0,C 180,E1 -1033.975,E2 -1033.975} C_VEL
LIN {X 0,Y 594.979,Z 478.438,A -85,B 0,C 180,E1 -1034.868,E2 -1034.868} C_VEL
LIN {X 0,Y 595.129,Z 462.696,A -85,B 0,C 180,E1 -1035.657,E2 -1035.657} C_VEL
LIN {X 0,Y 595.264,Z 447.61,A -85,B 0,C 180,E1 -1036.268,E2 -1036.268} C_VEL
LIN {X 0,Y 595.355,Z 430.954,A -85,B 0,C 180,E1 -1036.789,E2 -1036.789} C_VEL
LIN {X 0,Y 595.44,Z 413.865,A -85,B 0,C 180,E1 -1037.17,E2 -1037.17} C_VEL
LIN {X 0,Y 595.505,Z 382.628,A -85,B 0,C 180,E1 -1037.591,E2 -1037.591} C_VEL
LIN {X 0,Y 595.768,Z 209.56,A -85,B 0,C 180,E1 -1039.78,E2 -1039.78} C_VEL
LIN {X 0,Y 595.128,Z 205.851,A -85,B 0,C 180,E1 -1039.857,E2 -1039.857} C_VEL
LIN {X 0,Y 595.097,Z 186.651,A -85,B 0,C 180,E1 -1041.682,E2 -1041.682} C_VEL
LIN {X 0,Y 594.385,Z 183.761,A -85,B 0,C 180,E1 -1042.005,E2 -1042.005} C_VEL
LIN {X 0,Y 594.361,Z 183.761,A -85,B 0,C 180,E1 -1044.675,E2 -1044.675} C_VEL
LIN {X 0,Y 594.379,Z 183.754,A -85,B 0,C 180,E1 -1047.088,E2 -1047.088} C_VEL
LIN {X 0,Y 594.386,Z 183.755,A -85,B 0,C 180,E1 -1049.671,E2 -1049.671} C_VEL
LIN {X 0,Y 594.374,Z 183.758,A -85,B 0,C 180,E1 -1052.539,E2 -1052.539} C_VEL
LIN {X 0,Y 594.372,Z 183.756,A -85,B 0,C 180,E1 -1054.806,E2 -1054.806} C_VEL
LIN {X 0,Y 594.363,Z 183.756,A -85,B 0,C 180,E1 -1057.264,E2 -1057.264} C_VEL
LIN {X 0,Y 594.372,Z 183.763,A -85,B 0,C 180,E1 -1059.946,E2 -1059.946} C_VEL
LIN {X 0,Y 594.386,Z 183.752,A -85,B 0,C 180,E1 -1062.806,E2 -1062.806} C_VEL
LIN {X 0,Y 594.386,Z 183.761,A -85,B 0,C 180,E1 -1065.826,E2 -1065.826} C_VEL
LIN {X 0,Y 594.389,Z 183.755,A -85,B 0,C 180,E1 -1068.404,E2 -1068.404} C_VEL
LIN {X 0,Y 594.377,Z 183.754,A -85,B 0,C 180,E1 -1071.157,E2 -1071.157} C_VEL
LIN {X 0,Y 594.361,Z 183.765,A -85,B 0,C 180,E1 -1073.891,E2 -1073.891} C_VEL
LIN {X 0,Y 594.37,Z 183.754,A -85,B 0,C 180,E1 -1076.61,E2 -1076.61} C_VEL
LIN {X 0,Y 594.422,Z 183.752,A -85,B 0,C 180,E1 -1079.322,E2 -1079.322} C_VEL
LIN {X 0,Y 594.382,Z 183.757,A -85,B 0,C 180,E1 -1082.032,E2 -1082.032} C_VEL
LIN {X 0,Y 594.378,Z 183.753,A -85,B 0,C 180,E1 -1084.747,E2 -1084.747} C_VEL
LIN {X 0,Y 594.398,Z 183.759,A -85,B 0,C 180,E1 -1087.473,E2 -1087.473} C_VEL
LIN {X 0,Y 594.38,Z 183.754,A -85,B 0,C 180,E1 -1090.216,E2 -1090.216} C_VEL
LIN {X 0,Y 594.358,Z 183.758,A -85,B 0,C 180,E1 -1092.983,E2 -1092.983} C_VEL
LIN {X 0,Y 594.366,Z 183.759,A -85,B 0,C 180,E1 -1095.078,E2 -1095.078} C_VEL
LIN {X 0,Y 594.384,Z 183.759,A -85,B 0,C 180,E1 -1097.193,E2 -1097.193} C_VEL
LIN {X 0,Y 594.363,Z 183.756,A -85,B 0,C 180,E1 -1100.054,E2 -1100.054} C_VEL
LIN {X 0,Y 594.359,Z 183.76,A -85,B 0,C 180,E1 -1102.967,E2 -1102.967} C_VEL
LIN {X 0,Y 594.366,Z 183.763,A -85,B 0,C 180,E1 -1105.193,E2 -1105.193} C_VEL
LIN {X 0,Y 594.382,Z 183.759,A -85,B 0,C 180,E1 -1107.527,E2 -1107.527} C_VEL
LIN {X 0,Y 594.365,Z 183.755,A -85,B 0,C 180,E1 -1110.325,E2 -1110.325} C_VEL
LIN {X 0,Y 594.373,Z 183.76,A -85,B 0,C 180,E1 -1112.95,E2 -1112.95} C_VEL
LIN {X 0,Y 594.345,Z 183.763,A -85,B 0,C 180,E1 -1115.409,E2 -1115.409} C_VEL
LIN {X 0,Y 594.373,Z 183.754,A -85,B 0,C 180,E1 -1117.941,E2 -1117.941} C_VEL
LIN {X 0,Y 594.371,Z 183.761,A -85,B 0,C 180,E1 -1120.821,E2 -1120.821} C_VEL
LIN {X 0,Y 594.349,Z 183.762,A -85,B 0,C 180,E1 -1123.301,E2 -1123.301} C_VEL
LIN {X 0,Y 594.358,Z 183.757,A -85,B 0,C 180,E1 -1126.161,E2 -1126.161} C_VEL
LIN {X 0,Y 594.373,Z 183.76,A -85,B 0,C 180,E1 -1129.178,E2 -1129.178} C_VEL
LIN {X 0,Y 594.371,Z 183.755,A -85,B 0,C 180,E1 -1132.058,E2 -1132.058} C_VEL
LIN {X 0,Y 594.348,Z 183.766,A -85,B 0,C 180,E1 -1134.677,E2 -1134.677} C_VEL
LIN {X 0,Y 594.372,Z 183.759,A -85,B 0,C 180,E1 -1137.089,E2 -1137.089} C_VEL
LIN {X 0,Y 594.365,Z 183.756,A -85,B 0,C 180,E1 -1139.675,E2 -1139.675} C_VEL
LIN {X 0,Y 594.376,Z 183.763,A -85,B 0,C 180,E1 -1142.539,E2 -1142.539} C_VEL
LIN {X 0,Y 594.404,Z 183.936,A -85,B 0,C 180,E1 -1142.826,E2 -1142.826} C_VEL
LIN {X 0,Y 595.513,Z 188.353,A -85,B 0,C 180,E1 -1143.26,E2 -1143.26} C_VEL
LIN {X 0,Y 595.307,Z 220.372,A -85,B 0,C 180,E1 -1145.964,E2 -1145.964} C_VEL
LIN {X 0,Y 595.192,Z 235.005,A -85,B 0,C 180,E1 -1147.181,E2 -1147.181} C_VEL
LIN {X 0,Y 595.791,Z 238.598,A -85,B 0,C 180,E1 -1147.254,E2 -1147.254} C_VEL
LIN {X 0,Y 595.464,Z 442.372,A -85,B 0,C 180,E1 -1149.849,E2 -1149.849} C_VEL
LIN {X 0,Y 595.387,Z 458.05,A -85,B 0,C 180,E1 -1150.183,E2 -1150.183} C_VEL
LIN {X 0,Y 595.272,Z 473.915,A -85,B 0,C 180,E1 -1150.65,E2 -1150.65} C_VEL
LIN {X 0,Y 595.156,Z 489.464,A -85,B 0,C 180,E1 -1151.244,E2 -1151.244} C_VEL
LIN {X 0,Y 595.057,Z 503.997,A -85,B 0,C 180,E1 -1151.938,E2 -1151.938} C_VEL
LIN {X 0,Y 594.896,Z 517.83,A -85,B 0,C 180,E1 -1152.732,E2 -1152.732} C_VEL
LIN {X 0,Y 594.802,Z 532.039,A -85,B 0,C 180,E1 -1153.702,E2 -1153.702} C_VEL
LIN {X 0,Y 594.648,Z 545.113,A -85,B 0,C 180,E1 -1154.753,E2 -1154.753} C_VEL
LIN {X 0,Y 594.561,Z 557.304,A -85,B 0,C 180,E1 -1155.903,E2 -1155.903} C_VEL
LIN {X 0,Y 594.449,Z 568.9,A -85,B 0,C 180,E1 -1157.191,E2 -1157.191} C_VEL
LIN {X 0,Y 594.383,Z 579.416,A -85,B 0,C 180,E1 -1158.573,E2 -1158.573} C_VEL
LIN {X 0,Y 594.334,Z 588.265,A -85,B 0,C 180,E1 -1159.954,E2 -1159.954} C_VEL
LIN {X 0,Y 594.295,Z 596.481,A -85,B 0,C 180,E1 -1161.498,E2 -1161.498} C_VEL
LIN {X 0,Y 594.285,Z 602.462,A -85,B 0,C 180,E1 -1162.866,E2 -1162.866} C_VEL
LIN {X 0,Y 594.264,Z 608.242,A -85,B 0,C 180,E1 -1164.57,E2 -1164.57} C_VEL
LIN {X 0,Y 594.252,Z 611.631,A -85,B 0,C 180,E1 -1165.929,E2 -1165.929} C_VEL
LIN {X 0,Y 594.213,Z 614.085,A -85,B 0,C 180,E1 -1167.287,E2 -1167.287} C_VEL
LIN {X 0,Y 594.24,Z 615.477,A -85,B 0,C 180,E1 -1168.643,E2 -1168.643} C_VEL
LIN {X 0,Y 594.231,Z 616,A -85,B 0,C 180,E1 -1169.998,E2 -1169.998} C_VEL
LIN {X 0,Y 594.24,Z 615.479,A -85,B 0,C 180,E1 -1171.354,E2 -1171.354} C_VEL
LIN {X 0,Y 594.213,Z 614.089,A -85,B 0,C 180,E1 -1172.71,E2 -1172.71} C_VEL
LIN {X 0,Y 594.252,Z 611.638,A -85,B 0,C 180,E1 -1174.067,E2 -1174.067} C_VEL
LIN {X 0,Y 594.281,Z 607.191,A -85,B 0,C 180,E1 -1175.767,E2 -1175.767} C_VEL
LIN {X 0,Y 594.287,Z 602.476,A -85,B 0,C 180,E1 -1177.131,E2 -1177.131} C_VEL
LIN {X 0,Y 594.317,Z 594.867,A -85,B 0,C 180,E1 -1178.841,E2 -1178.841} C_VEL
LIN {X 0,Y 594.354,Z 586.26,A -85,B 0,C 180,E1 -1180.387,E2 -1180.387} C_VEL
LIN {X 0,Y 594.405,Z 576.985,A -85,B 0,C 180,E1 -1181.766,E2 -1181.766} C_VEL
LIN {X 0,Y 594.468,Z 567.442,A -85,B 0,C 180,E1 -1182.979,E2 -1182.979} C_VEL
LIN {X 0,Y 594.534,Z 555.971,A -85,B 0,C 180,E1 -1184.229,E2 -1184.229} C_VEL
LIN {X 0,Y 594.676,Z 544.169,A -85,B 0,C 180,E1 -1185.331,E2 -1185.331} C_VEL
LIN {X 0,Y 594.808,Z 530.913,A -85,B 0,C 180,E1 -1186.383,E2 -1186.383} C_VEL
LIN {X 0,Y 594.926,Z 516.473,A -85,B 0,C 180,E1 -1187.352,E2 -1187.352} C_VEL
LIN {X 0,Y 595.044,Z 502.315,A -85,B 0,C 180,E1 -1188.148,E2 -1188.148} C_VEL
LIN {X 0,Y 595.202,Z 486.954,A -85,B 0,C 180,E1 -1188.861,E2 -1188.861} C_VEL
LIN {X 0,Y 595.275,Z 471.418,A -85,B 0,C 180,E1 -1189.436,E2 -1189.436} C_VEL
LIN {X 0,Y 595.388,Z 455.455,A -85,B 0,C 180,E1 -1189.881,E2 -1189.881} C_VEL
LIN {X 0,Y 595.493,Z 439.604,A -85,B 0,C 180,E1 -1190.192,E2 -1190.192} C_VEL
LIN {X 0,Y 595.776,Z 238.627,A -85,B 0,C 180,E1 -1192.746,E2 -1192.746} C_VEL
LIN {X 0,Y 595.209,Z 234.822,A -85,B 0,C 180,E1 -1192.834,E2 -1192.834} C_VEL
LIN {X 0,Y 595.44,Z 201.645,A -85,B 0,C 180,E1 -1195.61,E2 -1195.61} C_VEL
LIN {X 0,Y 595.539,Z 188.395,A -85,B 0,C 180,E1 -1196.735,E2 -1196.735} C_VEL
LIN {X 0,Y 594.386,Z 183.763,A -85,B 0,C 180,E1 -1197.195,E2 -1197.195} C_VEL
LIN {X 0,Y 594.347,Z 183.761,A -85,B 0,C 180,E1 -1199.775,E2 -1199.775} C_VEL
LIN {X 0,Y 594.341,Z 183.758,A -85,B 0,C 180,E1 -1202.145,E2 -1202.145} C_VEL
LIN {X 0,Y 594.37,Z 183.756,A -85,B 0,C 180,E1 -1204.577,E2 -1204.577} C_VEL
LIN {X 0,Y 594.37,Z 183.759,A -85,B 0,C 180,E1 -1207.606,E2 -1207.606} C_VEL
LIN {X 0,Y 594.341,Z 183.759,A -85,B 0,C 180,E1 -1210.565,E2 -1210.565} C_VEL
LIN {X 0,Y 594.356,Z 183.765,A -85,B 0,C 180,E1 -1213.296,E2 -1213.296} C_VEL
LIN {X 0,Y 594.341,Z 183.757,A -85,B 0,C 180,E1 -1216.159,E2 -1216.159} C_VEL
LIN {X 0,Y 594.354,Z 183.758,A -85,B 0,C 180,E1 -1218.534,E2 -1218.534} C_VEL
LIN {X 0,Y 594.364,Z 183.762,A -85,B 0,C 180,E1 -1221.293,E2 -1221.293} C_VEL
LIN {X 0,Y 594.349,Z 183.757,A -85,B 0,C 180,E1 -1223.756,E2 -1223.756} C_VEL
LIN {X 0,Y 594.337,Z 183.759,A -85,B 0,C 180,E1 -1226.236,E2 -1226.236} C_VEL
LIN {X 0,Y 594.362,Z 183.758,A -85,B 0,C 180,E1 -1228.65,E2 -1228.65} C_VEL
LIN {X 0,Y 594.362,Z 183.765,A -85,B 0,C 180,E1 -1231.039,E2 -1231.039} C_VEL
LIN {X 0,Y 594.366,Z 183.758,A -85,B 0,C 180,E1 -1233.3,E2 -1233.3} C_VEL
LIN {X 0,Y 594.357,Z 183.757,A -85,B 0,C 180,E1 -1236.295,E2 -1236.295} C_VEL
LIN {X 0,Y 594.386,Z 183.756,A -85,B 0,C 180,E1 -1239.224,E2 -1239.224} C_VEL
LIN {X 0,Y 594.349,Z 183.757,A -85,B 0,C 180,E1 -1242.095,E2 -1242.095} C_VEL
LIN {X 0,Y 594.342,Z 183.759,A -85,B 0,C 180,E1 -1244.219,E2 -1244.219} C_VEL
LIN {X 0,Y 594.35,Z 183.761,A -85,B 0,C 180,E1 -1247.017,E2 -1247.017} C_VEL
LIN {X 0,Y 594.383,Z 183.757,A -85,B 0,C 180,E1 -1249.095,E2 -1249.095} C_VEL
LIN {X 0,Y 594.377,Z 183.753,A -85,B 0,C 180,E1 -1251.843,E2 -1251.843} C_VEL
LIN {X 0,Y 594.382,Z 183.76,A -85,B 0,C 180,E1 -1254.572,E2 -1254.572} C_VEL
LIN {X 0,Y 594.381,Z 183.753,A -85,B 0,C 180,E1 -1257.289,E2 -1257.289} C_VEL
LIN {X 0,Y 594.368,Z 183.755,A -85,B 0,C 180,E1 -1260,E2 -1260} C_VEL
LIN {X 0,Y 594.398,Z 183.76,A -85,B 0,C 180,E1 -1262.711,E2 -1262.711} C_VEL
LIN {X 0,Y 594.362,Z 183.755,A -85,B 0,C 180,E1 -1265.428,E2 -1265.428} C_VEL
LIN {X 0,Y 594.382,Z 183.756,A -85,B 0,C 180,E1 -1268.158,E2 -1268.158} C_VEL
LIN {X 0,Y 594.373,Z 183.755,A -85,B 0,C 180,E1 -1271.085,E2 -1271.085} C_VEL
LIN {X 0,Y 594.348,Z 183.757,A -85,B 0,C 180,E1 -1273.68,E2 -1273.68} C_VEL
LIN {X 0,Y 594.334,Z 183.759,A -85,B 0,C 180,E1 -1275.359,E2 -1275.359} C_VEL
LIN {X 0,Y 593.658,Z 183.845,A -85,B 0,C 180,E1 -1275.924,E2 -1275.924} C_VEL
LIN {X 0,Y 590.788,Z 184.204,A -85,B 0,C 180,E1 -1276.843,E2 -1276.843} C_VEL
LIN {X 0,Y 588.38,Z 184.505,A -85,B 0,C 180,E1 -1277.581,E2 -1277.581} C_VEL
LIN {X 0,Y 587.364,Z 184.63,A -85,B 0,C 180,E1 -1278.152,E2 -1278.152} C_VEL
LIN {X 0,Y 587.292,Z 184.638,A -85,B 0,C 180,E1 -1278.345,E2 -1278.345} C_VEL
LIN {X 0,Y 587.326,Z 184.633,A -85,B 0,C 180,E1 -1281.046,E2 -1281.046} C_VEL
LIN {X 0,Y 587.335,Z 184.631,A -85,B 0,C 180,E1 -1283.259,E2 -1283.259} C_VEL
LIN {X 0,Y 587.328,Z 184.636,A -85,B 0,C 180,E1 -1286.183,E2 -1286.183} C_VEL
LIN {X 0,Y 587.327,Z 184.632,A -85,B 0,C 180,E1 -1289.137,E2 -1289.137} C_VEL
LIN {X 0,Y 587.322,Z 184.634,A -85,B 0,C 180,E1 -1291.839,E2 -1291.839} C_VEL
LIN {X 0,Y 587.321,Z 184.642,A -85,B 0,C 180,E1 -1294.35,E2 -1294.35} C_VEL
LIN {X 0,Y 587.328,Z 184.635,A -85,B 0,C 180,E1 -1296.749,E2 -1296.749} C_VEL
LIN {X 0,Y 587.305,Z 184.632,A -85,B 0,C 180,E1 -1299.363,E2 -1299.363} C_VEL
LIN {X 0,Y 587.317,Z 184.641,A -85,B 0,C 180,E1 -1302.111,E2 -1302.111} C_VEL
LIN {X 0,Y 587.28,Z 184.636,A -85,B 0,C 180,E1 -1305.09,E2 -1305.09} C_VEL
LIN {X 0,Y 587.296,Z 184.641,A -85,B 0,C 180,E1 -1307.927,E2 -1307.927} C_VEL
LIN {X 0,Y 587.314,Z 184.635,A -85,B 0,C 180,E1 -1310.642,E2 -1310.642} C_VEL
LIN {X 0,Y 587.334,Z 184.631,A -85,B 0,C 180,E1 -1313.295,E2 -1313.295} C_VEL
LIN {X 0,Y 587.34,Z 184.634,A -85,B 0,C 180,E1 -1315.782,E2 -1315.782} C_VEL
LIN {X 0,Y 587.32,Z 184.64,A -85,B 0,C 180,E1 -1318.233,E2 -1318.233} C_VEL
LIN {X 0,Y 587.334,Z 184.631,A -85,B 0,C 180,E1 -1320.87,E2 -1320.87} C_VEL
LIN {X 0,Y 587.304,Z 184.641,A -85,B 0,C 180,E1 -1323.831,E2 -1323.831} C_VEL
LIN {X 0,Y 587.3,Z 184.635,A -85,B 0,C 180,E1 -1326.743,E2 -1326.743} C_VEL
LIN {X 0,Y 587.306,Z 184.64,A -85,B 0,C 180,E1 -1329.697,E2 -1329.697} C_VEL
LIN {X 0,Y 587.282,Z 184.646,A -85,B 0,C 180,E1 -1331.874,E2 -1331.874} C_VEL
LIN {X 0,Y 587.3,Z 184.636,A -85,B 0,C 180,E1 -1334.738,E2 -1334.738} C_VEL
LIN {X 0,Y 587.278,Z 184.638,A -85,B 0,C 180,E1 -1336.86,E2 -1336.86} C_VEL
LIN {X 0,Y 587.326,Z 184.639,A -85,B 0,C 180,E1 -1339.662,E2 -1339.662} C_VEL
LIN {X 0,Y 587.312,Z 184.636,A -85,B 0,C 180,E1 -1342.438,E2 -1342.438} C_VEL
LIN {X 0,Y 587.333,Z 184.632,A -85,B 0,C 180,E1 -1345.197,E2 -1345.197} C_VEL
LIN {X 0,Y 587.371,Z 184.635,A -85,B 0,C 180,E1 -1347.945,E2 -1347.945} C_VEL
LIN {X 0,Y 587.383,Z 184.634,A -85,B 0,C 180,E1 -1350.002,E2 -1350.002} C_VEL
LIN {X 0,Y 587.354,Z 184.646,A -85,B 0,C 180,E1 -1351.866,E2 -1351.866} C_VEL
LIN {X 0,Y 588.412,Z 189.628,A -85,B 0,C 180,E1 -1352.397,E2 -1352.397} C_VEL
LIN {X 0,Y 588.318,Z 206.155,A -85,B 0,C 180,E1 -1353.962,E2 -1353.962} C_VEL
LIN {X 0,Y 589.225,Z 211.039,A -85,B 0,C 180,E1 -1354.063,E2 -1354.063} C_VEL
LIN {X 0,Y 588.808,Z 411.424,A -85,B 0,C 180,E1 -1356.641,E2 -1356.641} C_VEL
LIN {X 0,Y 588.696,Z 428.486,A -85,B 0,C 180,E1 -1357.002,E2 -1357.002} C_VEL
LIN {X 0,Y 588.533,Z 444.913,A -85,B 0,C 180,E1 -1357.498,E2 -1357.498} C_VEL
LIN {X 0,Y 588.391,Z 459.576,A -85,B 0,C 180,E1 -1358.069,E2 -1358.069} C_VEL
LIN {X 0,Y 588.235,Z 475.563,A -85,B 0,C 180,E1 -1358.85,E2 -1358.85} C_VEL
LIN {X 0,Y 588.047,Z 490.196,A -85,B 0,C 180,E1 -1359.72,E2 -1359.72} C_VEL
LIN {X 0,Y 587.873,Z 503.754,A -85,B 0,C 180,E1 -1360.68,E2 -1360.68} C_VEL
LIN {X 0,Y 587.719,Z 516.409,A -85,B 0,C 180,E1 -1361.73,E2 -1361.73} C_VEL
LIN {X 0,Y 587.561,Z 529.041,A -85,B 0,C 180,E1 -1362.961,E2 -1362.961} C_VEL
LIN {X 0,Y 587.444,Z 540.58,A -85,B 0,C 180,E1 -1364.288,E2 -1364.288} C_VEL
LIN {X 0,Y 587.356,Z 550.393,A -85,B 0,C 180,E1 -1365.619,E2 -1365.619} C_VEL
LIN {X 0,Y 587.257,Z 559.303,A -85,B 0,C 180,E1 -1367.053,E2 -1367.053} C_VEL
LIN {X 0,Y 587.228,Z 566.732,A -85,B 0,C 180,E1 -1368.492,E2 -1368.492} C_VEL
LIN {X 0,Y 587.197,Z 572.914,A -85,B 0,C 180,E1 -1369.945,E2 -1369.945} C_VEL
LIN {X 0,Y 587.156,Z 577.826,A -85,B 0,C 180,E1 -1371.413,E2 -1371.413} C_VEL
LIN {X 0,Y 587.134,Z 581.421,A -85,B 0,C 180,E1 -1372.824,E2 -1372.824} C_VEL
LIN {X 0,Y 587.119,Z 584.367,A -85,B 0,C 180,E1 -1374.529,E2 -1374.529} C_VEL
LIN {X 0,Y 587.129,Z 585.834,A -85,B 0,C 180,E1 -1376.289,E2 -1376.289} C_VEL
LIN {X 0,Y 587.147,Z 585.828,A -85,B 0,C 180,E1 -1377.829,E2 -1377.829} C_VEL
LIN {X 0,Y 587.135,Z 584.56,A -85,B 0,C 180,E1 -1379.392,E2 -1379.392} C_VEL
LIN {X 0,Y 587.144,Z 582.021,A -85,B 0,C 180,E1 -1380.978,E2 -1380.978} C_VEL
LIN {X 0,Y 587.15,Z 578.086,A -85,B 0,C 180,E1 -1382.591,E2 -1382.591} C_VEL
LIN {X 0,Y 587.197,Z 574.086,A -85,B 0,C 180,E1 -1383.818,E2 -1383.818} C_VEL
LIN {X 0,Y 587.245,Z 568.15,A -85,B 0,C 180,E1 -1385.293,E2 -1385.293} C_VEL
LIN {X 0,Y 587.271,Z 560.908,A -85,B 0,C 180,E1 -1386.753,E2 -1386.753} C_VEL
LIN {X 0,Y 587.311,Z 552.643,A -85,B 0,C 180,E1 -1388.13,E2 -1388.13} C_VEL
LIN {X 0,Y 587.433,Z 542.342,A -85,B 0,C 180,E1 -1389.575,E2 -1389.575} C_VEL
LIN {X 0,Y 587.535,Z 531.222,A -85,B 0,C 180,E1 -1390.893,E2 -1390.893} C_VEL
LIN {X 0,Y 587.683,Z 518.769,A -85,B 0,C 180,E1 -1392.145,E2 -1392.145} C_VEL
LIN {X 0,Y 587.837,Z 505.543,A -85,B 0,C 180,E1 -1393.273,E2 -1393.273} C_VEL
LIN {X 0,Y 588.026,Z 491.88,A -85,B 0,C 180,E1 -1394.261,E2 -1394.261} C_VEL
LIN {X 0,Y 588.214,Z 476.783,A -85,B 0,C 180,E1 -1395.175,E2 -1395.175} C_VEL
LIN {X 0,Y 588.375,Z 461.369,A -85,B 0,C 180,E1 -1395.94,E2 -1395.94} C_VEL
LIN {X 0,Y 588.538,Z 445.58,A -85,B 0,C 180,E1 -1396.569,E2 -1396.569} C_VEL
LIN {X 0,Y 588.702,Z 428.675,A -85,B 0,C 180,E1 -1397.083,E2 -1397.083} C_VEL
LIN {X 0,Y 588.795,Z 411.65,A -85,B 0,C 180,E1 -1397.445,E2 -1397.445} C_VEL
LIN {X 0,Y 589.251,Z 210.833,A -85,B 0,C 180,E1 -1400.029,E2 -1400.029} C_VEL
LIN {X 0,Y 588.35,Z 205.75,A -85,B 0,C 180,E1 -1400.144,E2 -1400.144} C_VEL
LIN {X 0,Y 588.379,Z 188.788,A -85,B 0,C 180,E1 -1401.775,E2 -1401.775} C_VEL
LIN {X 0,Y 587.366,Z 184.634,A -85,B 0,C 180,E1 -1402.24,E2 -1402.24} C_VEL
LIN {X 0,Y 587.334,Z 184.634,A -85,B 0,C 180,E1 -1404.944,E2 -1404.944} C_VEL
LIN {X 0,Y 587.339,Z 184.632,A -85,B 0,C 180,E1 -1407.42,E2 -1407.42} C_VEL
LIN {X 0,Y 587.334,Z 184.636,A -85,B 0,C 180,E1 -1409.829,E2 -1409.829} C_VEL
LIN {X 0,Y 587.352,Z 184.637,A -85,B 0,C 180,E1 -1412.306,E2 -1412.306} C_VEL
LIN {X 0,Y 587.332,Z 184.637,A -85,B 0,C 180,E1 -1414.483,E2 -1414.483} C_VEL
LIN {X 0,Y 587.317,Z 184.634,A -85,B 0,C 180,E1 -1417.131,E2 -1417.131} C_VEL
LIN {X 0,Y 587.328,Z 184.636,A -85,B 0,C 180,E1 -1419.695,E2 -1419.695} C_VEL
LIN {X 0,Y 587.354,Z 184.63,A -85,B 0,C 180,E1 -1422.594,E2 -1422.594} C_VEL
LIN {X 0,Y 587.362,Z 184.634,A -85,B 0,C 180,E1 -1425.739,E2 -1425.739} C_VEL
LIN {X 0,Y 587.345,Z 184.63,A -85,B 0,C 180,E1 -1428.866,E2 -1428.866} C_VEL
LIN {X 0,Y 587.361,Z 184.636,A -85,B 0,C 180,E1 -1431.744,E2 -1431.744} C_VEL
LIN {X 0,Y 587.348,Z 184.63,A -85,B 0,C 180,E1 -1434.507,E2 -1434.507} C_VEL
LIN {X 0,Y 587.373,Z 184.629,A -85,B 0,C 180,E1 -1437.256,E2 -1437.256} C_VEL
LIN {X 0,Y 587.374,Z 184.632,A -85,B 0,C 180,E1 -1440,E2 -1440} C_VEL
LIN {X 0,Y 587.364,Z 184.627,A -85,B 0,C 180,E1 -1442.743,E2 -1442.743} C_VEL
LIN {X 0,Y 587.355,Z 184.636,A -85,B 0,C 180,E1 -1445.493,E2 -1445.493} C_VEL
LIN {X 0,Y 587.335,Z 184.632,A -85,B 0,C 180,E1 -1448.255,E2 -1448.255} C_VEL
LIN {X 0,Y 587.344,Z 184.633,A -85,B 0,C 180,E1 -1451.133,E2 -1451.133} C_VEL
LIN {X 0,Y 587.351,Z 184.629,A -85,B 0,C 180,E1 -1454.257,E2 -1454.257} C_VEL
LIN {X 0,Y 587.343,Z 184.64,A -85,B 0,C 180,E1 -1457.406,E2 -1457.406} C_VEL
LIN {X 0,Y 587.32,Z 184.633,A -85,B 0,C 180,E1 -1460.305,E2 -1460.305} C_VEL
LIN {X 0,Y 587.315,Z 184.642,A -85,B 0,C 180,E1 -1463.259,E2 -1463.259} C_VEL
LIN {X 0,Y 587.322,Z 184.639,A -85,B 0,C 180,E1 -1465.517,E2 -1465.517} C_VEL
LIN {X 0,Y 587.342,Z 184.632,A -85,B 0,C 180,E1 -1467.818,E2 -1467.818} C_VEL
LIN {X 0,Y 587.321,Z 184.633,A -85,B 0,C 180,E1 -1470.508,E2 -1470.508} C_VEL
LIN {X 0,Y 587.333,Z 184.64,A -85,B 0,C 180,E1 -1473.111,E2 -1473.111} C_VEL
LIN {X 0,Y 587.286,Z 184.637,A -85,B 0,C 180,E1 -1475.9,E2 -1475.9} C_VEL
LIN {X 0,Y 587.317,Z 184.635,A -85,B 0,C 180,E1 -1478.48,E2 -1478.48} C_VEL
LIN {X 0,Y 587.33,Z 184.639,A -85,B 0,C 180,E1 -1481.157,E2 -1481.157} C_VEL
LIN {X 0,Y 587.3,Z 184.635,A -85,B 0,C 180,E1 -1484.111,E2 -1484.111} C_VEL
LIN {X 0,Y 587.297,Z 184.645,A -85,B 0,C 180,E1 -1486.992,E2 -1486.992} C_VEL
LIN {X 0,Y 587.309,Z 184.635,A -85,B 0,C 180,E1 -1489.745,E2 -1489.745} C_VEL
LIN {X 0,Y 587.34,Z 184.634,A -85,B 0,C 180,E1 -1492.392,E2 -1492.392} C_VEL
LIN {X 0,Y 587.338,Z 184.631,A -85,B 0,C 180,E1 -1495.653,E2 -1495.653} C_VEL
LIN {X 0,Y 587.332,Z 184.634,A -85,B 0,C 180,E1 -1498.23,E2 -1498.23} C_VEL
LIN {X 0,Y 587.341,Z 184.64,A -85,B 0,C 180,E1 -1500.868,E2 -1500.868} C_VEL
LIN {X 0,Y 587.357,Z 184.816,A -85,B 0,C 180,E1 -1502.549,E2 -1502.549} C_VEL
LIN {X 0,Y 588.676,Z 189.457,A -85,B 0,C 180,E1 -1503.02,E2 -1503.02} C_VEL
LIN {X 0,Y 588.837,Z 200.498,A -85,B 0,C 180,E1 -1503.983,E2 -1503.983} C_VEL
LIN {X 0,Y 588.482,Z 234.997,A -85,B 0,C 180,E1 -1506.905,E2 -1506.905} C_VEL
LIN {X 0,Y 589.251,Z 240.594,A -85,B 0,C 180,E1 -1507.013,E2 -1507.013} C_VEL
LIN {X 0,Y 588.791,Z 440.876,A -85,B 0,C 180,E1 -1509.587,E2 -1509.587} C_VEL
LIN {X 0,Y 588.707,Z 457.139,A -85,B 0,C 180,E1 -1509.926,E2 -1509.926} C_VEL
LIN {X 0,Y 588.532,Z 473.916,A -85,B 0,C 180,E1 -1510.42,E2 -1510.42} C_VEL
LIN {X 0,Y 588.409,Z 489.7,A -85,B 0,C 180,E1 -1511.032,E2 -1511.032} C_VEL
LIN {X 0,Y 588.25,Z 504.001,A -85,B 0,C 180,E1 -1511.722,E2 -1511.722} C_VEL
LIN {X 0,Y 588.063,Z 517.833,A -85,B 0,C 180,E1 -1512.525,E2 -1512.525} C_VEL
LIN {X 0,Y 587.87,Z 532.038,A -85,B 0,C 180,E1 -1513.504,E2 -1513.504} C_VEL
LIN {X 0,Y 587.73,Z 545.111,A -85,B 0,C 180,E1 -1514.569,E2 -1514.569} C_VEL
LIN {X 0,Y 587.566,Z 556.615,A -85,B 0,C 180,E1 -1515.662,E2 -1515.662} C_VEL
LIN {X 0,Y 587.449,Z 567.414,A -85,B 0,C 180,E1 -1516.86,E2 -1516.86} C_VEL
LIN {X 0,Y 587.354,Z 578.201,A -85,B 0,C 180,E1 -1518.262,E2 -1518.262} C_VEL
LIN {X 0,Y 587.297,Z 587.254,A -85,B 0,C 180,E1 -1519.658,E2 -1519.658} C_VEL
LIN {X 0,Y 587.246,Z 594.85,A -85,B 0,C 180,E1 -1521.048,E2 -1521.048} C_VEL
LIN {X 0,Y 587.209,Z 602.462,A -85,B 0,C 180,E1 -1522.779,E2 -1522.779} C_VEL
LIN {X 0,Y 587.188,Z 608.242,A -85,B 0,C 180,E1 -1524.504,E2 -1524.504} C_VEL
LIN {X 0,Y 587.167,Z 611.632,A -85,B 0,C 180,E1 -1525.88,E2 -1525.88} C_VEL
LIN {X 0,Y 587.119,Z 614.085,A -85,B 0,C 180,E1 -1527.254,E2 -1527.254} C_VEL
LIN {X 0,Y 587.14,Z 615.477,A -85,B 0,C 180,E1 -1528.627,E2 -1528.627} C_VEL
LIN {X 0,Y 587.132,Z 616,A -85,B 0,C 180,E1 -1529.998,E2 -1529.998} C_VEL
LIN {X 0,Y 587.14,Z 615.479,A -85,B 0,C 180,E1 -1531.37,E2 -1531.37} C_VEL
LIN {X 0,Y 587.119,Z 614.09,A -85,B 0,C 180,E1 -1532.743,E2 -1532.743} C_VEL
LIN {X 0,Y 587.167,Z 611.638,A -85,B 0,C 180,E1 -1534.116,E2 -1534.116} C_VEL
LIN {X 0,Y 587.188,Z 607.192,A -85,B 0,C 180,E1 -1535.837,E2 -1535.837} C_VEL
LIN {X 0,Y 587.21,Z 602.476,A -85,B 0,C 180,E1 -1537.217,E2 -1537.217} C_VEL
LIN {X 0,Y 587.244,Z 594.867,A -85,B 0,C 180,E1 -1538.948,E2 -1538.948} C_VEL
LIN {X 0,Y 587.301,Z 586.261,A -85,B 0,C 180,E1 -1540.513,E2 -1540.513} C_VEL
LIN {X 0,Y 587.364,Z 576.987,A -85,B 0,C 180,E1 -1541.909,E2 -1541.909} C_VEL
LIN {X 0,Y 587.448,Z 567.443,A -85,B 0,C 180,E1 -1543.136,E2 -1543.136} C_VEL
LIN {X 0,Y 587.584,Z 555.589,A -85,B 0,C 180,E1 -1544.439,E2 -1544.439} C_VEL
LIN {X 0,Y 587.768,Z 543.124,A -85,B 0,C 180,E1 -1545.604,E2 -1545.604} C_VEL
LIN {X 0,Y 587.908,Z 529.737,A -85,B 0,C 180,E1 -1546.67,E2 -1546.67} C_VEL
LIN {X 0,Y 588.084,Z 515.045,A -85,B 0,C 180,E1 -1547.65,E2 -1547.65} C_VEL
LIN {X 0,Y 588.286,Z 500.571,A -85,B 0,C 180,E1 -1548.454,E2 -1548.454} C_VEL
LIN {X 0,Y 588.467,Z 485.371,A -85,B 0,C 180,E1 -1549.149,E2 -1549.149} C_VEL
LIN {X 0,Y 588.611,Z 469.335,A -85,B 0,C 180,E1 -1549.733,E2 -1549.733} C_VEL
LIN {X 0,Y 588.747,Z 452.706,A -85,B 0,C 180,E1 -1550.183,E2 -1550.183} C_VEL
LIN {X 0,Y 588.809,Z 436.592,A -85,B 0,C 180,E1 -1550.477,E2 -1550.477} C_VEL
LIN {X 0,Y 589.252,Z 239.54,A -85,B 0,C 180,E1 -1553.001,E2 -1553.001} C_VEL
LIN {X 0,Y 588.464,Z 234.823,A -85,B 0,C 180,E1 -1553.111,E2 -1553.111} C_VEL
LIN {X 0,Y 588.817,Z 201.645,A -85,B 0,C 180,E1 -1555.919,E2 -1555.919} C_VEL
LIN {X 0,Y 588.887,Z 191.385,A -85,B 0,C 180,E1 -1556.802,E2 -1556.802} C_VEL
LIN {X 0,Y 588.06,Z 187.305,A -85,B 0,C 180,E1 -1557.198,E2 -1557.198} C_VEL
LIN {X 0,Y 587.329,Z 184.642,A -85,B 0,C 180,E1 -1557.475,E2 -1557.475} C_VEL
LIN {X 0,Y 587.302,Z 184.636,A -85,B 0,C 180,E1 -1560.169,E2 -1560.169} C_VEL
LIN {X 0,Y 587.317,Z 184.633,A -85,B 0,C 180,E1 -1562.577,E2 -1562.577} C_VEL
LIN {X 0,Y 587.314,Z 184.641,A -85,B 0,C 180,E1 -1565.053,E2 -1565.053} C_VEL
LIN {X 0,Y 587.316,Z 184.635,A -85,B 0,C 180,E1 -1567.836,E2 -1567.836} C_VEL
LIN {X 0,Y 587.294,Z 184.636,A -85,B 0,C 180,E1 -1570.252,E2 -1570.252} C_VEL
LIN {X 0,Y 587.301,Z 184.644,A -85,B 0,C 180,E1 -1573.117,E2 -1573.117} C_VEL
LIN {X 0,Y 587.297,Z 184.635,A -85,B 0,C 180,E1 -1576.047,E2 -1576.047} C_VEL
LIN {X 0,Y 587.315,Z 184.64,A -85,B 0,C 180,E1 -1578.922,E2 -1578.922} C_VEL
LIN {X 0,Y 587.308,Z 184.638,A -85,B 0,C 180,E1 -1581.519,E2 -1581.519} C_VEL
LIN {X 0,Y 587.319,Z 184.634,A -85,B 0,C 180,E1 -1584.453,E2 -1584.453} C_VEL
LIN {X 0,Y 587.309,Z 184.642,A -85,B 0,C 180,E1 -1586.886,E2 -1586.886} C_VEL
LIN {X 0,Y 587.312,Z 184.636,A -85,B 0,C 180,E1 -1589.487,E2 -1589.487} C_VEL
LIN {X 0,Y 587.32,Z 184.634,A -85,B 0,C 180,E1 -1592.305,E2 -1592.305} C_VEL
LIN {X 0,Y 587.319,Z 184.638,A -85,B 0,C 180,E1 -1595.24,E2 -1595.24} C_VEL
LIN {X 0,Y 587.336,Z 184.632,A -85,B 0,C 180,E1 -1597.486,E2 -1597.486} C_VEL
LIN {X 0,Y 587.316,Z 184.634,A -85,B 0,C 180,E1 -1600.424,E2 -1600.424} C_VEL
LIN {X 0,Y 587.319,Z 184.636,A -85,B 0,C 180,E1 -1603.311,E2 -1603.311} C_VEL
LIN {X 0,Y 587.331,Z 184.631,A -85,B 0,C 180,E1 -1606.154,E2 -1606.154} C_VEL
LIN {X 0,Y 587.376,Z 184.632,A -85,B 0,C 180,E1 -1608.963,E2 -1608.963} C_VEL
LIN {X 0,Y 587.333,Z 184.631,A -85,B 0,C 180,E1 -1611.745,E2 -1611.745} C_VEL
LIN {X 0,Y 587.342,Z 184.635,A -85,B 0,C 180,E1 -1614.507,E2 -1614.507} C_VEL
LIN {X 0,Y 587.347,Z 184.629,A -85,B 0,C 180,E1 -1617.257,E2 -1617.257} C_VEL
LIN {X 0,Y 587.338,Z 184.631,A -85,B 0,C 180,E1 -1620,E2 -1620} C_VEL
LIN {X 0,Y 587.361,Z 184.635,A -85,B 0,C 180,E1 -1622.744,E2 -1622.744} C_VEL
LIN {X 0,Y 587.326,Z 184.631,A -85,B 0,C 180,E1 -1625.494,E2 -1625.494} C_VEL
LIN {X 0,Y 587.338,Z 184.635,A -85,B 0,C 180,E1 -1628.256,E2 -1628.256} C_VEL
LIN {X 0,Y 587.346,Z 184.629,A -85,B 0,C 180,E1 -1631.152,E2 -1631.152} C_VEL
LIN {X 0,Y 587.33,Z 184.636,A -85,B 0,C 180,E1 -1634.262,E2 -1634.262} C_VEL
LIN {X 0,Y 587.32,Z 184.632,A -85,B 0,C 180,E1 -1637.407,E2 -1637.407} C_VEL
LIN {X 0,Y 587.292,Z 184.638,A -85,B 0,C 180,E1 -1638.345,E2 -1638.345} C_VEL
LIN {X 0,Y 586.656,Z 184.718,A -85,B 0,C 180,E1 -1638.917,E2 -1638.917} C_VEL
LIN {X 0,Y 583.822,Z 185.069,A -85,B 0,C 180,E1 -1639.845,E2 -1639.845} C_VEL
LIN {X 0,Y 581.403,Z 185.378,A -85,B 0,C 180,E1 -1640.592,E2 -1640.592} C_VEL
LIN {X 0,Y 580.35,Z 185.502,A -85,B 0,C 180,E1 -1641.169,E2 -1641.169} C_VEL
LIN {X 0,Y 580.258,Z 185.512,A -85,B 0,C 180,E1 -1641.364,E2 -1641.364} C_VEL
LIN {X 0,Y 580.271,Z 185.51,A -85,B 0,C 180,E1 -1643.559,E2 -1643.559} C_VEL
LIN {X 0,Y 580.262,Z 185.519,A -85,B 0,C 180,E1 -1646.336,E2 -1646.336} C_VEL
LIN {X 0,Y 580.272,Z 185.512,A -85,B 0,C 180,E1 -1648.978,E2 -1648.978} C_VEL
LIN {X 0,Y 580.279,Z 185.514,A -85,B 0,C 180,E1 -1652.034,E2 -1652.034} C_VEL
LIN {X 0,Y 580.264,Z 185.516,A -85,B 0,C 180,E1 -1654.699,E2 -1654.699} C_VEL
LIN {X 0,Y 580.275,Z 185.51,A -85,B 0,C 180,E1 -1657.271,E2 -1657.271} C_VEL
LIN {X 0,Y 580.275,Z 185.518,A -85,B 0,C 180,E1 -1660.274,E2 -1660.274} C_VEL
LIN {X 0,Y 580.263,Z 185.515,A -85,B 0,C 180,E1 -1662.708,E2 -1662.708} C_VEL
LIN {X 0,Y 580.238,Z 185.514,A -85,B 0,C 180,E1 -1665.613,E2 -1665.613} C_VEL
LIN {X 0,Y 580.256,Z 185.522,A -85,B 0,C 180,E1 -1668.233,E2 -1668.233} C_VEL
LIN {X 0,Y 580.255,Z 185.512,A -85,B 0,C 180,E1 -1670.967,E2 -1670.967} C_VEL
LIN {X 0,Y 580.258,Z 185.515,A -85,B 0,C 180,E1 -1673.599,E2 -1673.599} C_VEL
LIN {X 0,Y 580.299,Z 185.516,A -85,B 0,C 180,E1 -1676.148,E2 -1676.148} C_VEL
LIN {X 0,Y 580.257,Z 185.514,A -85,B 0,C 180,E1 -1678.617,E2 -1678.617} C_VEL
LIN {X 0,Y 580.275,Z 185.51,A -85,B 0,C 180,E1 -1681.026,E2 -1681.026} C_VEL
LIN {X 0,Y 580.258,Z 185.52,A -85,B 0,C 180,E1 -1684.152,E2 -1684.152} C_VEL
LIN {X 0,Y 580.251,Z 185.513,A -85,B 0,C 180,E1 -1687.002,E2 -1687.002} C_VEL
LIN {X 0,Y 580.251,Z 185.516,A -85,B 0,C 180,E1 -1689.439,E2 -1689.439} C_VEL
LIN {X 0,Y 580.239,Z 185.519,A -85,B 0,C 180,E1 -1691.647,E2 -1691.647} C_VEL
LIN {X 0,Y 580.268,Z 185.513,A -85,B 0,C 180,E1 -1694.549,E2 -1694.549} C_VEL
LIN {X 0,Y 580.241,Z 185.515,A -85,B 0,C 180,E1 -1696.697,E2 -1696.697} C_VEL
LIN {X 0,Y 580.307,Z 185.507,A -85,B 0,C 180,E1 -1698.829,E2 -1698.829} C_VEL
LIN {X 0,Y 580.303,Z 185.514,A -85,B 0,C 180,E1 -1701.646,E2 -1701.646} C_VEL
LIN {X 0,Y 580.3,Z 185.508,A -85,B 0,C 180,E1 -1704.442,E2 -1704.442} C_VEL
LIN {X 0,Y 580.311,Z 185.509,A -85,B 0,C 180,E1 -1707.225,E2 -1707.225} C_VEL
LIN {X 0,Y 580.351,Z 185.51,A -85,B 0,C 180,E1 -1710.002,E2 -1710.002} C_VEL
LIN {X 0,Y 580.302,Z 185.558,A -85,B 0,C 180,E1 -1711.628,E2 -1711.628} C_VEL
LIN {X 0,Y 581.642,Z 191.27,A -85,B 0,C 180,E1 -1712.252,E2 -1712.252} C_VEL
LIN {X 0,Y 581.548,Z 205.762,A -85,B 0,C 180,E1 -1713.661,E2 -1713.661} C_VEL
LIN {X 0,Y 582.686,Z 212.226,A -85,B 0,C 180,E1 -1713.805,E2 -1713.805} C_VEL
LIN {X 0,Y 582.165,Z 411.007,A -85,B 0,C 180,E1 -1716.391,E2 -1716.391} C_VEL
LIN {X 0,Y 582.022,Z 427.675,A -85,B 0,C 180,E1 -1716.741,E2 -1716.741} C_VEL
LIN {X 0,Y 581.831,Z 444.091,A -85,B 0,C 180,E1 -1717.233,E2 -1717.233} C_VEL
LIN {X 0,Y 581.653,Z 460.165,A -85,B 0,C 180,E1 -1717.867,E2 -1717.867} C_VEL
LIN {X 0,Y 581.43,Z 475.083,A -85,B 0,C 180,E1 -1718.604,E2 -1718.604} C_VEL
LIN {X 0,Y 581.224,Z 489.791,A -85,B 0,C 180,E1 -1719.484,E2 -1719.484} C_VEL
LIN {X 0,Y 580.992,Z 503.436,A -85,B 0,C 180,E1 -1720.455,E2 -1720.455} C_VEL
LIN {X 0,Y 580.768,Z 516.615,A -85,B 0,C 180,E1 -1721.561,E2 -1721.561} C_VEL
LIN {X 0,Y 580.583,Z 528.823,A -85,B 0,C 180,E1 -1722.764,E2 -1722.764} C_VEL
LIN {X 0,Y 580.426,Z 539.66,A -85,B 0,C 180,E1 -1724.016,E2 -1724.016} C_VEL
LIN {X 0,Y 580.322,Z 550.215,A -85,B 0,C 180,E1 -1725.453,E2 -1725.453} C_VEL
LIN {X 0,Y 580.19,Z 559.143,A -85,B 0,C 180,E1 -1726.902,E2 -1726.902} C_VEL
LIN {X 0,Y 580.158,Z 566.608,A -85,B 0,C 180,E1 -1728.36,E2 -1728.36} C_VEL
LIN {X 0,Y 580.124,Z 572.814,A -85,B 0,C 180,E1 -1729.83,E2 -1729.83} C_VEL
LIN {X 0,Y 580.072,Z 577.737,A -85,B 0,C 180,E1 -1731.315,E2 -1731.315} C_VEL
LIN {X 0,Y 580.051,Z 581.79,A -85,B 0,C 180,E1 -1732.951,E2 -1732.951} C_VEL
LIN {X 0,Y 580.01,Z 584.552,A -85,B 0,C 180,E1 -1734.662,E2 -1734.662} C_VEL
LIN {X 0,Y 580.049,Z 585.835,A -85,B 0,C 180,E1 -1736.284,E2 -1736.284} C_VEL
LIN {X 0,Y 580.048,Z 585.834,A -85,B 0,C 180,E1 -1737.811,E2 -1737.811} C_VEL
LIN {X 0,Y 580.072,Z 584.732,A -85,B 0,C 180,E1 -1739.268,E2 -1739.268} C_VEL
LIN {X 0,Y 580.065,Z 582.761,A -85,B 0,C 180,E1 -1740.657,E2 -1740.657} C_VEL
LIN {X 0,Y 580.07,Z 579.281,A -85,B 0,C 180,E1 -1742.215,E2 -1742.215} C_VEL
LIN {X 0,Y 580.104,Z 574.2,A -85,B 0,C 180,E1 -1743.869,E2 -1743.869} C_VEL
LIN {X 0,Y 580.13,Z 569.317,A -85,B 0,C 180,E1 -1745.131,E2 -1745.131} C_VEL
LIN {X 0,Y 580.199,Z 561.994,A -85,B 0,C 180,E1 -1746.663,E2 -1746.663} C_VEL
LIN {X 0,Y 580.264,Z 553.392,A -85,B 0,C 180,E1 -1748.149,E2 -1748.149} C_VEL
LIN {X 0,Y 580.394,Z 543.904,A -85,B 0,C 180,E1 -1749.524,E2 -1749.524} C_VEL
LIN {X 0,Y 580.53,Z 533.363,A -85,B 0,C 180,E1 -1750.824,E2 -1750.824} C_VEL
LIN {X 0,Y 580.694,Z 521.401,A -85,B 0,C 180,E1 -1752.082,E2 -1752.082} C_VEL
LIN {X 0,Y 580.905,Z 507.798,A -85,B 0,C 180,E1 -1753.292,E2 -1753.292} C_VEL
LIN {X 0,Y 581.15,Z 493.001,A -85,B 0,C 180,E1 -1754.396,E2 -1754.396} C_VEL
LIN {X 0,Y 581.375,Z 478.051,A -85,B 0,C 180,E1 -1755.323,E2 -1755.323} C_VEL
LIN {X 0,Y 581.602,Z 462.94,A -85,B 0,C 180,E1 -1756.096,E2 -1756.096} C_VEL
LIN {X 0,Y 581.843,Z 447.655,A -85,B 0,C 180,E1 -1756.727,E2 -1756.727} C_VEL
LIN {X 0,Y 582.004,Z 431.182,A -85,B 0,C 180,E1 -1757.255,E2 -1757.255} C_VEL
LIN {X 0,Y 582.143,Z 414.481,A -85,B 0,C 180,E1 -1757.638,E2 -1757.638} C_VEL
LIN {X 0,Y 582.238,Z 388.003,A -85,B 0,C 180,E1 -1758.011,E2 -1758.011} C_VEL
LIN {X 0,Y 582.666,Z 211.23,A -85,B 0,C 180,E1 -1760.299,E2 -1760.299} C_VEL
LIN {X 0,Y 581.608,Z 205.676,A -85,B 0,C 180,E1 -1760.435,E2 -1760.435} C_VEL
LIN {X 0,Y 581.736,Z 192.17,A -85,B 0,C 180,E1 -1761.745,E2 -1761.745} C_VEL
LIN {X 0,Y 580.315,Z 185.513,A -85,B 0,C 180,E1 -1762.487,E2 -1762.487} C_VEL
LIN {X 0,Y 580.301,Z 185.509,A -85,B 0,C 180,E1 -1765.441,E2 -1765.441} C_VEL
LIN {X 0,Y 580.303,Z 185.514,A -85,B 0,C 180,E1 -1767.969,E2 -1767.969} C_VEL
LIN {X 0,Y 580.303,Z 185.51,A -85,B 0,C 180,E1 -1770.69,E2 -1770.69} C_VEL
LIN {X 0,Y 580.291,Z 185.512,A -85,B 0,C 180,E1 -1773.666,E2 -1773.666} C_VEL
LIN {X 0,Y 580.3,Z 185.512,A -85,B 0,C 180,E1 -1775.683,E2 -1775.683} C_VEL
LIN {X 0,Y 580.271,Z 185.52,A -85,B 0,C 180,E1 -1777.947,E2 -1777.947} C_VEL
LIN {X 0,Y 580.299,Z 185.508,A -85,B 0,C 180,E1 -1780.913,E2 -1780.913} C_VEL
LIN {X 0,Y 580.277,Z 185.517,A -85,B 0,C 180,E1 -1783.825,E2 -1783.825} C_VEL
LIN {X 0,Y 580.322,Z 185.514,A -85,B 0,C 180,E1 -1785.983,E2 -1785.983} C_VEL
LIN {X 0,Y 580.302,Z 185.507,A -85,B 0,C 180,E1 -1788.826,E2 -1788.826} C_VEL
LIN {X 0,Y 580.324,Z 185.511,A -85,B 0,C 180,E1 -1791.643,E2 -1791.643} C_VEL
LIN {X 0,Y 580.314,Z 185.507,A -85,B 0,C 180,E1 -1794.44,E2 -1794.44} C_VEL
LIN {X 0,Y 580.338,Z 185.504,A -85,B 0,C 180,E1 -1797.223,E2 -1797.223} C_VEL
LIN {X 0,Y 580.343,Z 185.507,A -85,B 0,C 180,E1 -1800,E2 -1800} C_VEL
LIN {X 0,Y 580.331,Z 185.504,A -85,B 0,C 180,E1 -1802.776,E2 -1802.776} C_VEL
LIN {X 0,Y 580.319,Z 185.514,A -85,B 0,C 180,E1 -1805.559,E2 -1805.559} C_VEL
LIN {X 0,Y 580.304,Z 185.507,A -85,B 0,C 180,E1 -1808.356,E2 -1808.356} C_VEL
LIN {X 0,Y 580.296,Z 185.512,A -85,B 0,C 180,E1 -1811.191,E2 -1811.191} C_VEL
LIN {X 0,Y 580.312,Z 185.508,A -85,B 0,C 180,E1 -1814.017,E2 -1814.017} C_VEL
LIN {X 0,Y 580.308,Z 185.508,A -85,B 0,C 180,E1 -1816.914,E2 -1816.914} C_VEL
LIN {X 0,Y 580.281,Z 185.513,A -85,B 0,C 180,E1 -1819.823,E2 -1819.823} C_VEL
LIN {X 0,Y 580.264,Z 185.512,A -85,B 0,C 180,E1 -1822.053,E2 -1822.053} C_VEL
LIN {X 0,Y 580.299,Z 185.513,A -85,B 0,C 180,E1 -1825.08,E2 -1825.08} C_VEL
LIN {X 0,Y 580.294,Z 185.508,A -85,B 0,C 180,E1 -1828.185,E2 -1828.185} C_VEL
LIN {X 0,Y 580.273,Z 185.513,A -85,B 0,C 180,E1 -1830.693,E2 -1830.693} C_VEL
LIN {X 0,Y 580.28,Z 185.517,A -85,B 0,C 180,E1 -1833.313,E2 -1833.313} C_VEL
LIN {X 0,Y 580.241,Z 185.516,A -85,B 0,C 180,E1 -1835.756,E2 -1835.756} C_VEL
LIN {X 0,Y 580.281,Z 185.51,A -85,B 0,C 180,E1 -1838.147,E2 -1838.147} C_VEL
LIN {X 0,Y 580.293,Z 185.515,A -85,B 0,C 180,E1 -1840.844,E2 -1840.844} C_VEL
LIN {X 0,Y 580.24,Z 185.516,A -85,B 0,C 180,E1 -1843.661,E2 -1843.661} C_VEL
LIN {X 0,Y 580.266,Z 185.517,A -85,B 0,C 180,E1 -1846.61,E2 -1846.61} C_VEL
LIN {X 0,Y 580.288,Z 185.509,A -85,B 0,C 180,E1 -1849.73,E2 -1849.73} C_VEL
LIN {X 0,Y 580.286,Z 185.518,A -85,B 0,C 180,E1 -1852.73,E2 -1852.73} C_VEL
LIN {X 0,Y 580.29,Z 185.511,A -85,B 0,C 180,E1 -1855.442,E2 -1855.442} C_VEL
LIN {X 0,Y 580.284,Z 185.51,A -85,B 0,C 180,E1 -1857.972,E2 -1857.972} C_VEL
LIN {X 0,Y 580.275,Z 185.52,A -85,B 0,C 180,E1 -1860.695,E2 -1860.695} C_VEL
LIN {X 0,Y 580.262,Z 185.551,A -85,B 0,C 180,E1 -1862.262,E2 -1862.262} C_VEL
LIN {X 0,Y 582.179,Z 192.674,A -85,B 0,C 180,E1 -1862.977,E2 -1862.977} C_VEL
LIN {X 0,Y 581.93,Z 220.408,A -85,B 0,C 180,E1 -1865.378,E2 -1865.378} C_VEL
LIN {X 0,Y 581.754,Z 235.025,A -85,B 0,C 180,E1 -1866.624,E2 -1866.624} C_VEL
LIN {X 0,Y 582.741,Z 241.419,A -85,B 0,C 180,E1 -1866.752,E2 -1866.752} C_VEL
LIN {X 0,Y 582.16,Z 442.371,A -85,B 0,C 180,E1 -1869.367,E2 -1869.367} C_VEL
LIN {X 0,Y 582.05,Z 458.966,A -85,B 0,C 180,E1 -1869.732,E2 -1869.732} C_VEL
LIN {X 0,Y 581.827,Z 475.215,A -85,B 0,C 180,E1 -1870.231,E2 -1870.231} C_VEL
LIN {X 0,Y 581.606,Z 492.027,A -85,B 0,C 180,E1 -1870.909,E2 -1870.909} C_VEL
LIN {X 0,Y 581.415,Z 507.284,A -85,B 0,C 180,E1 -1871.682,E2 -1871.682} C_VEL
LIN {X 0,Y 581.192,Z 521.768,A -85,B 0,C 180,E1 -1872.566,E2 -1872.566} C_VEL
LIN {X 0,Y 580.949,Z 535.528,A -85,B 0,C 180,E1 -1873.573,E2 -1873.573} C_VEL
LIN {X 0,Y 580.744,Z 547.06,A -85,B 0,C 180,E1 -1874.558,E2 -1874.558} C_VEL
LIN {X 0,Y 580.592,Z 558.61,A -85,B 0,C 180,E1 -1875.698,E2 -1875.698} C_VEL
LIN {X 0,Y 580.413,Z 570.325,A -85,B 0,C 180,E1 -1877.054,E2 -1877.054} C_VEL
LIN {X 0,Y 580.318,Z 580.667,A -85,B 0,C 180,E1 -1878.472,E2 -1878.472} C_VEL
LIN {X 0,Y 580.219,Z 589.278,A -85,B 0,C 180,E1 -1879.883,E2 -1879.883} C_VEL
LIN {X 0,Y 580.165,Z 596.482,A -85,B 0,C 180,E1 -1881.289,E2 -1881.289} C_VEL
LIN {X 0,Y 580.12,Z 602.462,A -85,B 0,C 180,E1 -1882.691,E2 -1882.691} C_VEL
LIN {X 0,Y 580.112,Z 608.242,A -85,B 0,C 180,E1 -1884.437,E2 -1884.437} C_VEL
LIN {X 0,Y 580.085,Z 611.632,A -85,B 0,C 180,E1 -1885.83,E2 -1885.83} C_VEL
LIN {X 0,Y 580.031,Z 614.086,A -85,B 0,C 180,E1 -1887.22,E2 -1887.22} C_VEL
LIN {X 0,Y 580.04,Z 615.478,A -85,B 0,C 180,E1 -1888.61,E2 -1888.61} C_VEL
LIN {X 0,Y 580.033,Z 616,A -85,B 0,C 180,E1 -1889.998,E2 -1889.998} C_VEL
LIN {X 0,Y 580.04,Z 615.48,A -85,B 0,C 180,E1 -1891.387,E2 -1891.387} C_VEL
LIN {X 0,Y 580.031,Z 614.09,A -85,B 0,C 180,E1 -1892.776,E2 -1892.776} C_VEL
LIN {X 0,Y 580.085,Z 611.639,A -85,B 0,C 180,E1 -1894.167,E2 -1894.167} C_VEL
LIN {X 0,Y 580.099,Z 607.193,A -85,B 0,C 180,E1 -1895.909,E2 -1895.909} C_VEL
LIN {X 0,Y 580.12,Z 602.476,A -85,B 0,C 180,E1 -1897.306,E2 -1897.306} C_VEL
LIN {X 0,Y 580.178,Z 594.867,A -85,B 0,C 180,E1 -1899.058,E2 -1899.058} C_VEL
LIN {X 0,Y 580.24,Z 586.262,A -85,B 0,C 180,E1 -1900.642,E2 -1900.642} C_VEL
LIN {X 0,Y 580.333,Z 576.988,A -85,B 0,C 180,E1 -1902.056,E2 -1902.056} C_VEL
LIN {X 0,Y 580.439,Z 567.442,A -85,B 0,C 180,E1 -1903.298,E2 -1903.298} C_VEL
LIN {X 0,Y 580.629,Z 555.948,A -85,B 0,C 180,E1 -1904.58,E2 -1904.58} C_VEL
LIN {X 0,Y 580.818,Z 544.169,A -85,B 0,C 180,E1 -1905.706,E2 -1905.706} C_VEL
LIN {X 0,Y 581.002,Z 530.907,A -85,B 0,C 180,E1 -1906.784,E2 -1906.784} C_VEL
LIN {X 0,Y 581.231,Z 516.468,A -85,B 0,C 180,E1 -1907.774,E2 -1907.774} C_VEL
LIN {X 0,Y 581.475,Z 502.321,A -85,B 0,C 180,E1 -1908.587,E2 -1908.587} C_VEL
LIN {X 0,Y 581.703,Z 487.092,A -85,B 0,C 180,E1 -1909.31,E2 -1909.31} C_VEL
LIN {X 0,Y 581.9,Z 471.416,A -85,B 0,C 180,E1 -1909.901,E2 -1909.901} C_VEL
LIN {X 0,Y 582.047,Z 455.454,A -85,B 0,C 180,E1 -1910.356,E2 -1910.356} C_VEL
LIN {X 0,Y 582.187,Z 439.603,A -85,B 0,C 180,E1 -1910.674,E2 -1910.674} C_VEL
LIN {X 0,Y 582.692,Z 240.159,A -85,B 0,C 180,E1 -1913.267,E2 -1913.267} C_VEL
LIN {X 0,Y 581.747,Z 234.972,A -85,B 0,C 180,E1 -1913.38,E2 -1913.38} C_VEL
LIN {X 0,Y 582.175,Z 201.645,A -85,B 0,C 180,E1 -1916.237,E2 -1916.237} C_VEL
LIN {X 0,Y 582.183,Z 192.7,A -85,B 0,C 180,E1 -1917.02,E2 -1917.02} C_VEL
LIN {X 0,Y 580.297,Z 185.516,A -85,B 0,C 180,E1 -1917.764,E2 -1917.764} C_VEL
LIN {X 0,Y 580.265,Z 185.515,A -85,B 0,C 180,E1 -1920.692,E2 -1920.692} C_VEL
LIN {X 0,Y 580.287,Z 185.516,A -85,B 0,C 180,E1 -1923.314,E2 -1923.314} C_VEL
LIN {X 0,Y 580.23,Z 185.52,A -85,B 0,C 180,E1 -1925.754,E2 -1925.754} C_VEL
LIN {X 0,Y 580.265,Z 185.512,A -85,B 0,C 180,E1 -1928.144,E2 -1928.144} C_VEL
LIN {X 0,Y 580.278,Z 185.514,A -85,B 0,C 180,E1 -1930.841,E2 -1930.841} C_VEL
LIN {X 0,Y 580.258,Z 185.515,A -85,B 0,C 180,E1 -1933.655,E2 -1933.655} C_VEL
LIN {X 0,Y 580.259,Z 185.514,A -85,B 0,C 180,E1 -1936.606,E2 -1936.606} C_VEL
LIN {X 0,Y 580.279,Z 185.518,A -85,B 0,C 180,E1 -1939.155,E2 -1939.155} C_VEL
LIN {X 0,Y 580.263,Z 185.512,A -85,B 0,C 180,E1 -1941.925,E2 -1941.925} C_VEL
LIN {X 0,Y 580.275,Z 185.511,A -85,B 0,C 180,E1 -1944.455,E2 -1944.455} C_VEL
LIN {X 0,Y 580.262,Z 185.521,A -85,B 0,C 180,E1 -1946.974,E2 -1946.974} C_VEL
LIN {X 0,Y 580.273,Z 185.514,A -85,B 0,C 180,E1 -1949.424,E2 -1949.424} C_VEL
LIN {X 0,Y 580.289,Z 185.508,A -85,B 0,C 180,E1 -1952.135,E2 -1952.135} C_VEL
LIN {X 0,Y 580.288,Z 185.513,A -85,B 0,C 180,E1 -1955.268,E2 -1955.268} C_VEL
LIN {X 0,Y 580.256,Z 185.512,A -85,B 0,C 180,E1 -1957.947,E2 -1957.947} C_VEL
LIN {X 0,Y 580.302,Z 185.514,A -85,B 0,C 180,E1 -1960.914,E2 -1960.914} C_VEL
LIN {X 0,Y 580.25,Z 185.513,A -85,B 0,C 180,E1 -1963.825,E2 -1963.825} C_VEL
LIN {X 0,Y 580.255,Z 185.52,A -85,B 0,C 180,E1 -1966.696,E2 -1966.696} C_VEL
LIN {X 0,Y 580.354,Z 185.507,A -85,B 0,C 180,E1 -1968.828,E2 -1968.828} C_VEL
LIN {X 0,Y 580.299,Z 185.507,A -85,B 0,C 180,E1 -1971.644,E2 -1971.644} C_VEL
LIN {X 0,Y 580.304,Z 185.511,A -85,B 0,C 180,E1 -1974.44,E2 -1974.44} C_VEL
LIN {X 0,Y 580.314,Z 185.505,A -85,B 0,C 180,E1 -1977.224,E2 -1977.224} C_VEL
LIN {X 0,Y 580.308,Z 185.507,A -85,B 0,C 180,E1 -1980,E2 -1980} C_VEL
LIN {X 0,Y 580.324,Z 185.511,A -85,B 0,C 180,E1 -1982.777,E2 -1982.777} C_VEL
LIN {X 0,Y 580.291,Z 185.507,A -85,B 0,C 180,E1 -1985.56,E2 -1985.56} C_VEL
LIN {X 0,Y 580.303,Z 185.513,A -85,B 0,C 180,E1 -1988.357,E2 -1988.357} C_VEL
LIN {X 0,Y 580.299,Z 185.506,A -85,B 0,C 180,E1 -1991.209,E2 -1991.209} C_VEL
LIN {X 0,Y 580.292,Z 185.509,A -85,B 0,C 180,E1 -1994.018,E2 -1994.018} C_VEL
LIN {X 0,Y 580.312,Z 185.508,A -85,B 0,C 180,E1 -1996.926,E2 -1996.926} C_VEL
LIN {X 0,Y 580.281,Z 185.508,A -85,B 0,C 180,E1 -1999.824,E2 -1999.824} C_VEL
LIN {X 0,Y 580.258,Z 185.512,A -85,B 0,C 180,E1 -2001.364,E2 -2001.364} C_VEL
LIN {X 0,Y 579.57,Z 185.601,A -85,B 0,C 180,E1 -2001.944,E2 -2001.944} C_VEL
LIN {X 0,Y 576.697,Z 185.959,A -85,B 0,C 180,E1 -2002.884,E2 -2002.884} C_VEL
LIN {X 0,Y 574.298,Z 186.256,A -85,B 0,C 180,E1 -2003.64,E2 -2003.64} C_VEL
LIN {X 0,Y 573.294,Z 186.386,A -85,B 0,C 180,E1 -2004.225,E2 -2004.225} C_VEL
LIN {X 0,Y 573.225,Z 186.391,A -85,B 0,C 180,E1 -2004.422,E2 -2004.422} C_VEL
LIN {X 0,Y 573.222,Z 186.389,A -85,B 0,C 180,E1 -2006.978,E2 -2006.978} C_VEL
LIN {X 0,Y 573.221,Z 186.389,A -85,B 0,C 180,E1 -2009.491,E2 -2009.491} C_VEL
LIN {X 0,Y 573.23,Z 186.391,A -85,B 0,C 180,E1 -2012.647,E2 -2012.647} C_VEL
LIN {X 0,Y 573.228,Z 186.388,A -85,B 0,C 180,E1 -2015.187,E2 -2015.187} C_VEL
LIN {X 0,Y 573.212,Z 186.392,A -85,B 0,C 180,E1 -2017.81,E2 -2017.81} C_VEL
LIN {X 0,Y 573.248,Z 186.391,A -85,B 0,C 180,E1 -2020.531,E2 -2020.531} C_VEL
LIN {X 0,Y 573.217,Z 186.389,A -85,B 0,C 180,E1 -2023.362,E2 -2023.362} C_VEL
LIN {X 0,Y 573.216,Z 186.398,A -85,B 0,C 180,E1 -2026.335,E2 -2026.335} C_VEL
LIN {X 0,Y 573.208,Z 186.395,A -85,B 0,C 180,E1 -2028.545,E2 -2028.545} C_VEL
LIN {X 0,Y 573.221,Z 186.388,A -85,B 0,C 180,E1 -2031.301,E2 -2031.301} C_VEL
LIN {X 0,Y 573.226,Z 186.397,A -85,B 0,C 180,E1 -2034.017,E2 -2034.017} C_VEL
LIN {X 0,Y 573.258,Z 186.388,A -85,B 0,C 180,E1 -2036.521,E2 -2036.521} C_VEL
LIN {X 0,Y 573.213,Z 186.39,A -85,B 0,C 180,E1 -2039.122,E2 -2039.122} C_VEL
LIN {X 0,Y 573.212,Z 186.391,A -85,B 0,C 180,E1 -2041.437,E2 -2041.437} C_VEL
LIN {X 0,Y 573.227,Z 186.39,A -85,B 0,C 180,E1 -2044.592,E2 -2044.592} C_VEL
LIN {X 0,Y 573.213,Z 186.394,A -85,B 0,C 180,E1 -2047.664,E2 -2047.664} C_VEL
LIN {X 0,Y 573.266,Z 186.383,A -85,B 0,C 180,E1 -2050.734,E2 -2050.734} C_VEL
LIN {X 0,Y 573.205,Z 186.396,A -85,B 0,C 180,E1 -2053.623,E2 -2053.623} C_VEL
LIN {X 0,Y 573.255,Z 186.394,A -85,B 0,C 180,E1 -2055.809,E2 -2055.809} C_VEL
LIN {X 0,Y 573.265,Z 186.384,A -85,B 0,C 180,E1 -2058.747,E2 -2058.747} C_VEL
LIN {X 0,Y 573.245,Z 186.392,A -85,B 0,C 180,E1 -2061.542,E2 -2061.542} C_VEL
LIN {X 0,Y 573.269,Z 186.384,A -85,B 0,C 180,E1 -2064.374,E2 -2064.374} C_VEL
LIN {X 0,Y 573.31,Z 186.387,A -85,B 0,C 180,E1 -2067.894,E2 -2067.894} C_VEL
LIN {X 0,Y 573.32,Z 186.386,A -85,B 0,C 180,E1 -2070.002,E2 -2070.002} C_VEL
LIN {X 0,Y 573.262,Z 186.551,A -85,B 0,C 180,E1 -2071.385,E2 -2071.385} C_VEL
LIN {X 0,Y 574.873,Z 192.914,A -85,B 0,C 180,E1 -2072.103,E2 -2072.103} C_VEL
LIN {X 0,Y 574.796,Z 205.817,A -85,B 0,C 180,E1 -2073.375,E2 -2073.375} C_VEL
LIN {X 0,Y 576.169,Z 213.374,A -85,B 0,C 180,E1 -2073.542,E2 -2073.542} C_VEL
LIN {X 0,Y 575.544,Z 410.563,A -85,B 0,C 180,E1 -2076.135,E2 -2076.135} C_VEL
LIN {X 0,Y 575.358,Z 427.459,A -85,B 0,C 180,E1 -2076.489,E2 -2076.489} C_VEL
LIN {X 0,Y 575.162,Z 443.61,A -85,B 0,C 180,E1 -2076.976,E2 -2076.976} C_VEL
LIN {X 0,Y 574.945,Z 458.786,A -85,B 0,C 180,E1 -2077.574,E2 -2077.574} C_VEL
LIN {X 0,Y 574.62,Z 474.615,A -85,B 0,C 180,E1 -2078.352,E2 -2078.352} C_VEL
LIN {X 0,Y 574.378,Z 489.412,A -85,B 0,C 180,E1 -2079.243,E2 -2079.243} C_VEL
LIN {X 0,Y 574.092,Z 503.135,A -85,B 0,C 180,E1 -2080.226,E2 -2080.226} C_VEL
LIN {X 0,Y 573.87,Z 515.884,A -85,B 0,C 180,E1 -2081.301,E2 -2081.301} C_VEL
LIN {X 0,Y 573.601,Z 528.61,A -85,B 0,C 180,E1 -2082.562,E2 -2082.562} C_VEL
LIN {X 0,Y 573.42,Z 539.455,A -85,B 0,C 180,E1 -2083.829,E2 -2083.829} C_VEL
LIN {X 0,Y 573.283,Z 550.04,A -85,B 0,C 180,E1 -2085.283,E2 -2085.283} C_VEL
LIN {X 0,Y 573.144,Z 558.578,A -85,B 0,C 180,E1 -2086.675,E2 -2086.675} C_VEL
LIN {X 0,Y 573.078,Z 566.488,A -85,B 0,C 180,E1 -2088.224,E2 -2088.224} C_VEL
LIN {X 0,Y 573.059,Z 572.709,A -85,B 0,C 180,E1 -2089.711,E2 -2089.711} C_VEL
LIN {X 0,Y 572.993,Z 577.675,A -85,B 0,C 180,E1 -2091.223,E2 -2091.223} C_VEL
LIN {X 0,Y 572.948,Z 580.635,A -85,B 0,C 180,E1 -2092.351,E2 -2092.351} C_VEL
LIN {X 0,Y 572.92,Z 583.533,A -85,B 0,C 180,E1 -2093.88,E2 -2093.88} C_VEL
LIN {X 0,Y 572.918,Z 585.336,A -85,B 0,C 180,E1 -2095.427,E2 -2095.427} C_VEL
LIN {X 0,Y 572.94,Z 585.995,A -85,B 0,C 180,E1 -2096.992,E2 -2096.992} C_VEL
LIN {X 0,Y 572.934,Z 585.391,A -85,B 0,C 180,E1 -2098.582,E2 -2098.582} C_VEL
LIN {X 0,Y 572.946,Z 583.559,A -85,B 0,C 180,E1 -2100.194,E2 -2100.194} C_VEL
LIN {X 0,Y 572.955,Z 580.4,A -85,B 0,C 180,E1 -2101.834,E2 -2101.834} C_VEL
LIN {X 0,Y 573,Z 575.767,A -85,B 0,C 180,E1 -2103.501,E2 -2103.501} C_VEL
LIN {X 0,Y 573.066,Z 569.452,A -85,B 0,C 180,E1 -2105.198,E2 -2105.198} C_VEL
LIN {X 0,Y 573.129,Z 562.355,A -85,B 0,C 180,E1 -2106.713,E2 -2106.713} C_VEL
LIN {X 0,Y 573.225,Z 554.808,A -85,B 0,C 180,E1 -2108.058,E2 -2108.058} C_VEL
LIN {X 0,Y 573.336,Z 545.657,A -85,B 0,C 180,E1 -2109.442,E2 -2109.442} C_VEL
LIN {X 0,Y 573.494,Z 535.586,A -85,B 0,C 180,E1 -2110.735,E2 -2110.735} C_VEL
LIN {X 0,Y 573.692,Z 524.455,A -85,B 0,C 180,E1 -2111.96,E2 -2111.96} C_VEL
LIN {X 0,Y 573.92,Z 512.07,A -85,B 0,C 180,E1 -2113.127,E2 -2113.127} C_VEL
LIN {X 0,Y 574.216,Z 498.169,A -85,B 0,C 180,E1 -2114.238,E2 -2114.238} C_VEL
LIN {X 0,Y 574.47,Z 483.903,A -85,B 0,C 180,E1 -2115.2,E2 -2115.2} C_VEL
LIN {X 0,Y 574.76,Z 468.867,A -85,B 0,C 180,E1 -2116.042,E2 -2116.042} C_VEL
LIN {X 0,Y 575.043,Z 453.004,A -85,B 0,C 180,E1 -2116.76,E2 -2116.76} C_VEL
LIN {X 0,Y 575.252,Z 436.788,A -85,B 0,C 180,E1 -2117.337,E2 -2117.337} C_VEL
LIN {X 0,Y 575.447,Z 419.579,A -85,B 0,C 180,E1 -2117.785,E2 -2117.785} C_VEL
LIN {X 0,Y 575.58,Z 402.858,A -85,B 0,C 180,E1 -2118.071,E2 -2118.071} C_VEL
LIN {X 0,Y 576.156,Z 212.417,A -85,B 0,C 180,E1 -2120.561,E2 -2120.561} C_VEL
LIN {X 0,Y 574.828,Z 205.744,A -85,B 0,C 180,E1 -2120.721,E2 -2120.721} C_VEL
LIN {X 0,Y 574.958,Z 193.724,A -85,B 0,C 180,E1 -2121.902,E2 -2121.902} C_VEL
LIN {X 0,Y 573.28,Z 186.39,A -85,B 0,C 180,E1 -2122.749,E2 -2122.749} C_VEL
LIN {X 0,Y 573.272,Z 186.387,A -85,B 0,C 180,E1 -2125.671,E2 -2125.671} C_VEL
LIN {X 0,Y 573.241,Z 186.395,A -85,B 0,C 180,E1 -2128.184,E2 -2128.184} C_VEL
LIN {X 0,Y 573.266,Z 186.388,A -85,B 0,C 180,E1 -2130.634,E2 -2130.634} C_VEL
LIN {X 0,Y 573.25,Z 186.387,A -85,B 0,C 180,E1 -2133.024,E2 -2133.024} C_VEL
LIN {X 0,Y 573.274,Z 186.384,A -85,B 0,C 180,E1 -2135.366,E2 -2135.366} C_VEL
LIN {X 0,Y 573.228,Z 186.392,A -85,B 0,C 180,E1 -2138.419,E2 -2138.419} C_VEL
LIN {X 0,Y 573.277,Z 186.384,A -85,B 0,C 180,E1 -2140.728,E2 -2140.728} C_VEL
LIN {X 0,Y 573.249,Z 186.389,A -85,B 0,C 180,E1 -2143.621,E2 -2143.621} C_VEL
LIN {X 0,Y 573.27,Z 186.391,A -85,B 0,C 180,E1 -2145.807,E2 -2145.807} C_VEL
LIN {X 0,Y 573.26,Z 186.385,A -85,B 0,C 180,E1 -2148.745,E2 -2148.745} C_VEL
LIN {X 0,Y 573.28,Z 186.387,A -85,B 0,C 180,E1 -2151.54,E2 -2151.54} C_VEL
LIN {X 0,Y 573.282,Z 186.384,A -85,B 0,C 180,E1 -2154.371,E2 -2154.371} C_VEL
LIN {X 0,Y 573.3,Z 186.387,A -85,B 0,C 180,E1 -2157.892,E2 -2157.892} C_VEL
LIN {X 0,Y 573.325,Z 186.376,A -85,B 0,C 180,E1 -2160.702,E2 -2160.702} C_VEL
LIN {X 0,Y 573.234,Z 186.395,A -85,B 0,C 180,E1 -2163.514,E2 -2163.514} C_VEL
LIN {X 0,Y 573.285,Z 186.391,A -85,B 0,C 180,E1 -2165.628,E2 -2165.628} C_VEL
LIN {X 0,Y 573.27,Z 186.39,A -85,B 0,C 180,E1 -2167.75,E2 -2167.75} C_VEL
LIN {X 0,Y 573.259,Z 186.384,A -85,B 0,C 180,E1 -2170.596,E2 -2170.596} C_VEL
LIN {X 0,Y 573.256,Z 186.385,A -85,B 0,C 180,E1 -2172.748,E2 -2172.748} C_VEL
LIN {X 0,Y 573.229,Z 186.39,A -85,B 0,C 180,E1 -2174.92,E2 -2174.92} C_VEL
LIN {X 0,Y 573.236,Z 186.39,A -85,B 0,C 180,E1 -2177.848,E2 -2177.848} C_VEL
LIN {X 0,Y 573.236,Z 186.388,A -85,B 0,C 180,E1 -2180.077,E2 -2180.077} C_VEL
LIN {X 0,Y 573.23,Z 186.388,A -85,B 0,C 180,E1 -2182.338,E2 -2182.338} C_VEL
LIN {X 0,Y 573.243,Z 186.395,A -85,B 0,C 180,E1 -2185.41,E2 -2185.41} C_VEL
LIN {X 0,Y 573.247,Z 186.387,A -85,B 0,C 180,E1 -2188.029,E2 -2188.029} C_VEL
LIN {X 0,Y 573.221,Z 186.394,A -85,B 0,C 180,E1 -2190.881,E2 -2190.881} C_VEL
LIN {X 0,Y 573.238,Z 186.391,A -85,B 0,C 180,E1 -2193.52,E2 -2193.52} C_VEL
LIN {X 0,Y 573.211,Z 186.39,A -85,B 0,C 180,E1 -2196.051,E2 -2196.051} C_VEL
LIN {X 0,Y 573.235,Z 186.392,A -85,B 0,C 180,E1 -2198.702,E2 -2198.702} C_VEL
LIN {X 0,Y 573.224,Z 186.391,A -85,B 0,C 180,E1 -2201.592,E2 -2201.592} C_VEL
LIN {X 0,Y 573.215,Z 186.391,A -85,B 0,C 180,E1 -2204.335,E2 -2204.335} C_VEL
LIN {X 0,Y 573.222,Z 186.392,A -85,B 0,C 180,E1 -2207.36,E2 -2207.36} C_VEL
LIN {X 0,Y 573.24,Z 186.39,A -85,B 0,C 180,E1 -2210.392,E2 -2210.392} C_VEL
LIN {X 0,Y 573.231,Z 186.395,A -85,B 0,C 180,E1 -2213.076,E2 -2213.076} C_VEL
LIN {X 0,Y 573.259,Z 186.386,A -85,B 0,C 180,E1 -2215.67,E2 -2215.67} C_VEL
LIN {X 0,Y 573.225,Z 186.391,A -85,B 0,C 180,E1 -2218.183,E2 -2218.183} C_VEL
LIN {X 0,Y 573.24,Z 186.397,A -85,B 0,C 180,E1 -2220.632,E2 -2220.632} C_VEL
LIN {X 0,Y 573.241,Z 186.46,A -85,B 0,C 180,E1 -2221.994,E2 -2221.994} C_VEL
LIN {X 0,Y 575.458,Z 194.128,A -85,B 0,C 180,E1 -2222.782,E2 -2222.782} C_VEL
LIN {X 0,Y 575.305,Z 213.747,A -85,B 0,C 180,E1 -2224.492,E2 -2224.492} C_VEL
LIN {X 0,Y 575.036,Z 234.969,A -85,B 0,C 180,E1 -2226.33,E2 -2226.33} C_VEL
LIN {X 0,Y 576.211,Z 242.229,A -85,B 0,C 180,E1 -2226.483,E2 -2226.483} C_VEL
LIN {X 0,Y 575.506,Z 442.371,A -85,B 0,C 180,E1 -2229.118,E2 -2229.118} C_VEL
LIN {X 0,Y 575.352,Z 458.968,A -85,B 0,C 180,E1 -2229.486,E2 -2229.486} C_VEL
LIN {X 0,Y 575.109,Z 475.214,A -85,B 0,C 180,E1 -2229.99,E2 -2229.99} C_VEL
LIN {X 0,Y 574.885,Z 491.173,A -85,B 0,C 180,E1 -2230.637,E2 -2230.637} C_VEL
LIN {X 0,Y 574.663,Z 505.699,A -85,B 0,C 180,E1 -2231.366,E2 -2231.366} C_VEL
LIN {X 0,Y 574.364,Z 520.636,A -85,B 0,C 180,E1 -2232.277,E2 -2232.277} C_VEL
LIN {X 0,Y 574.055,Z 534.37,A -85,B 0,C 180,E1 -2233.278,E2 -2233.278} C_VEL
LIN {X 0,Y 573.832,Z 547.058,A -85,B 0,C 180,E1 -2234.368,E2 -2234.368} C_VEL
LIN {X 0,Y 573.607,Z 559.27,A -85,B 0,C 180,E1 -2235.594,E2 -2235.594} C_VEL
LIN {X 0,Y 573.419,Z 570.327,A -85,B 0,C 180,E1 -2236.893,E2 -2236.893} C_VEL
LIN {X 0,Y 573.285,Z 580.664,A -85,B 0,C 180,E1 -2238.329,E2 -2238.329} C_VEL
LIN {X 0,Y 573.168,Z 589.277,A -85,B 0,C 180,E1 -2239.757,E2 -2239.757} C_VEL
LIN {X 0,Y 573.077,Z 596.482,A -85,B 0,C 180,E1 -2241.181,E2 -2241.181} C_VEL
LIN {X 0,Y 573.041,Z 602.461,A -85,B 0,C 180,E1 -2242.6,E2 -2242.6} C_VEL
LIN {X 0,Y 573.016,Z 607.182,A -85,B 0,C 180,E1 -2244.014,E2 -2244.014} C_VEL
LIN {X 0,Y 573.006,Z 611.633,A -85,B 0,C 180,E1 -2245.778,E2 -2245.778} C_VEL
LIN {X 0,Y 572.947,Z 614.086,A -85,B 0,C 180,E1 -2247.186,E2 -2247.186} C_VEL
LIN {X 0,Y 572.94,Z 615.478,A -85,B 0,C 180,E1 -2248.593,E2 -2248.593} C_VEL
LIN {X 0,Y 572.933,Z 616,A -85,B 0,C 180,E1 -2249.998,E2 -2249.998} C_VEL
LIN {X 0,Y 572.939,Z 615.48,A -85,B 0,C 180,E1 -2251.404,E2 -2251.404} C_VEL
LIN {X 0,Y 572.946,Z 614.091,A -85,B 0,C 180,E1 -2252.811,E2 -2252.811} C_VEL
